FUNCTION_BLOCK FB_IndexedPatchPressMachine
VAR
    fbPatchFeedManager : FB_PatchFeedManager;
    bPatchDriveRunRequest : BOOL;
    bPatchSequenceAirRequest : BOOL;
    bPatchSequenceDownRequest : BOOL;
    bPatchHoldUpAllowed : BOOL;
    bPatchStartAllowed : BOOL;
    bPatchVerticalIndexReady : BOOL;
    bPatchVerticalUpCommandPrevious : BOOL;
    bPatchVerticalDownCommandPrevious : BOOL;
    fbIndex : FB_IndexTable4;
    fbMainDoorLock : FB_MainDoorLock;
    fbNestManager : FB_NestTableManager;
    fbOperatorStation : FB_OperatorStation;
    bOperatorLoadValid : BOOL;
    fbPatchDispense : FB_PatchDispenseStation;
    fbHeatStake : FB_HeatStakeStation;
    fbHeatStakeTemperature : FB_HeatStakeTemperatureControl;
    fbHeatStakePressureRegulator : FB_VeabPressureRegulator;
    fbVision : FB_VisionStation;
    fbVisionManualImages : FB_VisionManualImages;
    aVisionPbupReferenceKnown : ARRAY[1..4] OF BOOL;
    uiVisionPbupNest : UINT;
    uiVisionPbupEditNest : UINT;
    uiVisionImageOwnedNest : UINT;
    eVisionImageOwnedIndex : E_TablePosition;
    bVisionImagePermit : BOOL;
    bVisionImageJogBusy : BOOL;
    bVisionImageOwnedBeforeUpdate : BOOL;
    bVisionImageRecoveryRequired : BOOL;
    bManualImageTriggerCommand : BOOL;
    bManualCameraTransportReady : BOOL;
    bManualImageCameraFailed : BOOL;
    bVisionPbupFitted : BOOL;
    bVisionPbupKnown : BOOL;
    rtVisionPbupAutoBusy : R_TRIG;
    rtVisionPbupAutoDone : R_TRIG;
    tonVisionRotate0Confirm : TON;
    tonVisionRotate180Confirm : TON;
    tVisionRotaryConfirm : TIME := T#1S;
    bVisionRotate0Confirmed : BOOL;
    bVisionRotate180Confirmed : BOOL;
    bVisionRotate0CommandPrevious : BOOL;
    bVisionRotate180CommandPrevious : BOOL;
    bVisionTriggerAccepted : BOOL;
    bVisionRotatingCaptureAccepted : BOOL;
	fbVSCamera : FB_VSCamera;
    fbProcessCycle : FB_ProcessCycle;
    fbCommissioningGuard : FB_PatchPressCommissioningGuard;
    eMachineState : E_MachineState := E_MachineState.PowerUp;
    eInitialisingWaitReason : E_InitialisingWaitReason := E_InitialisingWaitReason.None;
    eStoppingWaitReason : E_StoppingWaitReason := E_StoppingWaitReason.None;
    stOutputsInternal : ST_MachineOutputs;
    stIndexStatus : ST_IndexStatus;
    stMainDoorStatus : ST_MainDoorLockStatus;
    stOperatorStatus : ST_OperatorStationStatus;
    stPatchDispenseStatus : ST_PatchStageStatus;
    stHeatStakeStatus : ST_PatchStageStatus;
    stHeatStakeTemperatureStatus : ST_HeatStakeTemperatureStatus;
    stHeatStakeProcessStatus : ST_HeatStakeProcessStatus;
    stVisionStatus : ST_PatchStageStatus;
    stOperatorNest : ST_Nest;
    stPatchDispenseNest : ST_Nest;
    stHeatStakeNest : ST_Nest;
    stHeatStakePresenceResult : ST_ProcessResult;
    stEmptyHeatStakePresenceResult : ST_ProcessResult;
    stVisionNest : ST_Nest;
	stPatchDispenseCycleResult : ST_ProcessResult;
    stHeatStakeCycleResult : ST_ProcessResult;

    bPatchDispenseRequired : BOOL;
    bHeatStakeRequired : BOOL;
    bVisionRequired : BOOL;
	
	bPatchHomeVerticalUpRequest : BOOL := FALSE;
	
	// Patch Dispensing Manual Mode
	bPatchManualEnableAllowed : BOOL;
	bPatchManualSupportAllowed : BOOL;
	bPatchManualVerticalAllowed : BOOL;
	bPatchManualAirAllowed : BOOL;

    // Snapshot taken before the station Update() calls.
    // Required to know which physical parts were actually being processed if
    // Safety is lost, because Update() immediately disables the station when
    // Safety_OK goes FALSE.
    bVisionProcessingBeforeUpdate 			: BOOL;

    // Machine-state transition tracking for one-shot product disposition.
    ePreviousMachineState 					: E_MachineState := E_MachineState.PowerUp;
    stProcessFaultResult 					: ST_ProcessResult;

    bAllRequiredStationsReady 				: BOOL;
    bAllRequiredStationsComplete 			: BOOL;
    bAnyStationInProcess 					: BOOL;
    bCycleResultsStored 					: BOOL;

    stPermissives 							: ST_MachinePermissives;
    tonInitialising 						: TON;
    tonStopping 							: TON;
	tonHeaterDwell 							: TON;

	
	
	bHeaterDwellTimeoutFault 				: BOOL := FALSE;
    bInitialisationTimeoutFault 			: BOOL;
    bStoppingTimeoutFault 					: BOOL;
    bAutoCycleAllowed 						: BOOL;
    sAutoCycleBlockReason 					: STRING(160);
    bIndexMoveAccepted 						: BOOL;
    bDoorLockOutput 						: BOOL;
	bMainDoorUnlockAcknowledged 			: BOOL := FALSE;
	bMainDoorHotLockRequired 				: BOOL := FALSE;
	
    rtManualIndexMove 						: R_TRIG;
	rtReprocessIndexAttempt 				: R_TRIG;
	rtMachineInitialising 					: R_TRIG;

    bProcessStartStations       			: BOOL;
    bProcessStopStations        			: BOOL;
    bProcessRequestIndex        			: BOOL;
    bProcessCycleActive         			: BOOL;
    bProcessCycleCompletePulse  			: BOOL;
    bProcessCycleFault          			: BOOL;
    bProcessCycleTimeoutFault   			: BOOL;
    bProcessStopPending         			: BOOL;
    bProcessAutomaticStopRequest 			: BOOL;
    bAutoCycleStopRequestLatched 			: BOOL;
    eProcessCycleState          			: E_CycleState;
    bDisabledNestIndexAttempt   			: BOOL;

    aNestSnapshot               			: ARRAY[1..4] OF ST_Nest;
    bDisabledNestPartPresent    			: BOOL;
    uiDisabledNestPartNestId    			: UINT;
    bDisabledNestPartPopupRequest 			: BOOL;
    uiDisabledNestPartPopupNestId 			: UINT;
    iNestCheck                  			: INT;

    // Reject chute full supervision / controlled stop.
    tonRejectChuteFull              : TON;
    tonRejectChutePopupReopen       : TON;
    rtRejectChuteAcknowledge        : R_TRIG;
    rtRejectChuteStopRequest        : R_TRIG;
    bRejectChuteFullLatched         : BOOL;
    bRejectChutePopupRequest        : BOOL;
    bRejectChuteStopRequestLatched  : BOOL;
    bRejectChutePopupReopenPending  : BOOL;
	bReprocessPopupAcknowledged 	: BOOL := FALSE;
	bReprocessAcknowledgePending 	: BOOL := FALSE;
	bHeaterDwellRequestLatched 		: BOOL := FALSE;

    // Manual controlled-stop tracking.
    bManualSupportTargetUpAtRejectStop : BOOL;
    bManualRejectStopReady             : BOOL;

    bStation1SupportExtendRequest  	: BOOL;
    bStation1SupportRetractRequest 	: BOOL;
    bStation2SupportExtendRequest  	: BOOL;
    bStation2SupportRetractRequest 	: BOOL;

    bHeatStakeHeadLockRequest 		: BOOL;
    bHeatStakeHeadUnlockRequest 	: BOOL;
    // Monostable valve output state; re-arm descent only after completed HOME.
    bHeatStakeHeadUpRecoveryLatched : BOOL := TRUE;
    bHeatStakeHeadDownHeld : BOOL := FALSE;
    bHeatStakeHeadDownRequest 		: BOOL;
    bHeatStakeHeadUpRequest 		: BOOL;
    rHeatStakePressureCommandBar 	: LREAL;
    iHeatStakePressureRaw 			: INT;
    rHeatStakePressureScaledBar 	: LREAL;
    bHeatStakeContactDwellActive 	: BOOL;
    usiHeatStakeSequenceStep 		: USINT;
	
	rtPatchSupportExtend 			: R_TRIG;
	rtPatchSupportRetract 			: R_TRIG;
	bPatchSupportExtendDesired 		: BOOL := FALSE;
	bPatchManualAllowed 			: BOOL;
	tpPatchAirBlow 					: TP;


    // Heat Stake Manual Mode
    rtHeatStakeManualStakePatch 	: R_TRIG;
    rtHeatStakeManualUnlock     	: R_TRIG;
    rtHeatStakeManualLock       	: R_TRIG;
    rtHeatStakeManualHeadDown   	: R_TRIG;
    rtHeatStakeManualHeadUp     	: R_TRIG;
    rtHeatStakeInitialising     	: R_TRIG;

    tonHeatStakeManualAction     	: TON;
    usiHeatStakeManualActionStep 	: USINT := 0;
    bHeatStakeManualHeadUnlocked 	: BOOL := FALSE;
    bHeatStakeManualStakeCycleActive : BOOL := FALSE;

    bHeatStakeStationHeadDownTimeoutFault 		: BOOL;
    bHeatStakeStationHeadUpTimeoutFault 		: BOOL;
    bHeatStakeStationHeadSensorConflictFault 	: BOOL;
    bHeatStakeManualHeadDownTimeoutFault 		: BOOL;
    bHeatStakeManualHeadUpTimeoutFault 			: BOOL;

    bHeatStakeManualEnableAllowed   : BOOL;
    bHeatStakeManualStakeAllowed    : BOOL;
    bHeatStakeManualUnlockAllowed   : BOOL;
    bHeatStakeManualLockAllowed     : BOOL;
    bHeatStakeManualHeadDownAllowed : BOOL;
    bHeatStakeManualHeadUpAllowed   : BOOL;
    bHeatStakeManualSupportAllowed  : BOOL;
    bHeatStakeManualActionBusy      : BOOL;
	
	// Vision Manual Mode

	tpVisionManualHorizontalBack  	: TP;
	tpVisionManualHorizontalFront 	: TP;
	


	
	rtVisionManualHorizontalBack  	: R_TRIG;
	rtVisionManualHorizontalFront 	: R_TRIG;
	rtVisionManualHome 				: R_TRIG;
	
	// Vision Manual - Vertical Intermediate


	
	bVisionManualVerticalUpActive 			: BOOL;

	bVisionManualVerticalFullDownActive     : BOOL;
	
	bVisionManualRotate0Active   			: BOOL;
	bVisionManualRotate180Active 			: BOOL;

    // Manual Heat Stake tooling-position tracking uses physical sensors.
    bHeatStakeManualHomePosition     		: BOOL;
    bHeatStakeManualOutOfHome        		: BOOL;

    bVisionHorizontalBackRequest  : BOOL;
    bVisionHorizontalFrontRequest : BOOL;
    bVisionVerticalUpRequest      : BOOL;
    bVisionVerticalDownRequest    : BOOL;

    bVisionGripCloseRequest       : BOOL;
    bVisionGripOpenRequest        : BOOL;
    bVisionRotate0Request         : BOOL;
    bVisionRotate180Request       : BOOL;
	
	//CAMERA
	bVisionTriggerRequest			: BOOL;
	bVisionChangeProgramRequest		: BOOL;
	bVisionGetResultsRequest		: BOOL;
	bVisionGetResultsReadyRequest	: BOOL;
	bVisionResetResultsRequest		: BOOL;
	bVisionAcknowledgeResultsRquest	: BOOL;
	nVisionProgramNumber			: UDINT;
	bVisionGetCurrentProgram		: UDINT;
	
	nVisionResults					: ST_VisionResults;
    rtVisionCameraResultsReset : R_TRIG;
	
		
		// Vision Manual Mode
	bVisionManualEnableAllowed          : BOOL;
    bVisionCameraStartBlocked : BOOL; // Live camera error/recovery latch; blocks new starts.
	
	bVisionHorizontalBackAllowed        : BOOL;
	bVisionHorizontalFrontAllowed       : BOOL;
	
	bVisionVerticalUpAllowed            : BOOL;

	bVisionVerticalFullDownAllowed      : BOOL;
	
	bVisionGripOpenAllowed              : BOOL;
	bVisionGripCloseAllowed             : BOOL;
	
	bVisionRotate0Allowed               : BOOL;
	bVisionRotate180Allowed             : BOOL;
	
	bVisionManualRunSequenceAllowed 	: BOOL;
	bVisionManualSequenceActive 		: BOOL;
	bVisionManualHomeAllowed 			: BOOL;
	bVisionManualHomeActive  			: BOOL;

// Already existed:
// bVisionSupportAllowed : BOOL;
    // Fault reset is latched because PRG_Events executes after PRG_Main.
    // The event manager may clear its fault latch on the same Reset scan,
    // therefore the machine must remember the request until the following scan.
    bFaultResetRequested 				: BOOL;
    bAirAndDoorEnable 					: BOOL;
    // Air can only be latched ON by System Initialising.
    // Once ON, it may remain ON through Stopping/Stopped while the main door
    // stays closed. Opening the door, or entering Fault, clears this latch.
    bAirSupplyLatched 					: BOOL;
    // PLC-originated machine faults pulse the TwinSAFE Run/Stop request low.
    // RunRequest is otherwise TRUE so TwinSAFE can execute and return Safety_OK.
    bSafetyDropRequest 					: BOOL;
    tpSafetyRunDrop 					: TP;
    tonLedBlink 						: TON;
    rtLedBlink 							: R_TRIG;
	
	tonHMIAliveOn  						: TON;
	tonHMIAliveOff 						: TON;
	bOutHMI        						: BOOL := TRUE;
	
	
	
    bLedBlinkState : BOOL;
	
	btest								: ARRAY [1..10] OF BOOL;
	ntest								: UDINT;
	
	sHeaterMinimum 						: STRING(32);
	sHeaterCurrent 						: STRING(32);
	
	// =====================================================
	// PATCH DISPENSING - MANUAL VERTICAL
	// =====================================================
    bPatchManualVerticalUpHeld : BOOL := TRUE; // Retain the selected UP direction while manual control is permitted.
    bPatchManualVerticalDownHeld : BOOL; // Retain the selected DOWN direction while manual control is permitted.
	
	bPatchVerticalUpAllowed   : BOOL;
	bPatchVerticalDownAllowed : BOOL;
	
	tonPatchHomeUpOutputVerify : TON;
	bPatchHomeUpOutputVerified : BOOL := FALSE;
	
    // Per-product volatile confidence/location; existing retained fitted array stays compatible.
    aVisionProductLocation : ARRAY[1..4] OF USINT; // 0 unknown, 1 nest, 2 legacy nest alias, 3 held; PBUP state is separate.
    aVisionPbupSource : ARRAY[1..4] OF USINT;
    aVisionLoadEmptySeen : ARRAY[1..4] OF BOOL;
    aVisionLoadCandidate : ARRAY[1..4] OF BOOL;
    uiVisionLoadObservedNest : UINT;
    tonVisionLoadEmpty : TON;
    tonVisionLoadPair : TON;
    bManualIndexAttempt : BOOL;
    bManualIndexStartAllowed : BOOL;
    bManualIndexWarningActive : BOOL;
    bManualIndexBlockVision : BOOL;
    bManualIndexBlockHeat : BOOL;
    bManualIndexBlockPatch : BOOL;
    bManualIndexBlockOther : BOOL;
    bManualCameraDrainResult : BOOL;
    bManualCameraDiscardedResult : BOOL;
    stManualCameraDiscardedResults : ST_VisionResults;
    bManualCameraRecoveryAllowed : BOOL;
    bManualCameraRecoveryActive : BOOL;
    bManualCameraRecoveryFailed : BOOL;
    bManualCameraCaptureAfterRecovery : BOOL;
    bManualCameraClearError0 : BOOL;
    bManualCameraClearError1 : BOOL;
    usiManualCameraRecoveryStep : USINT;
    udiManualCameraRecoveryImage : UDINT;
    udiManualCameraRecoveryError0 : UDINT;
    udiManualCameraRecoveryError1 : UDINT;
    tonManualCameraRecovery : TON;
    sManualCameraRecoveryMessage : STRING(160);
    bManualCameraResetOnly : BOOL;
    bManualCameraRecoveredPulse : BOOL;
END_VAR
VAR
    bManualCameraAllowed : BOOL;
    bManualCameraOwner : BOOL;
    bManualCameraReset : BOOL;
    bManualCameraConsume : BOOL;
    usiManualCameraStep : USINT;
    udiManualCameraProgram : UDINT;
    udiManualCameraSelection : UDINT;
    stManualCameraResults : ST_VisionResults;
    tonManualCamera : TON;
END_VAR

METHOD PUBLIC Cyclic
VAR_INPUT
    stInputs : ST_MachineInputs;
    stCommand : ST_MachineCommand;
    stConfig : ST_MachineConfig;
    stHeatStakeTemperatureSettings : ST_HeatStakeTemperatureSettings;
    stHeatStakeProcessSettings : ST_HeatStakeProcessSettings;
    bPatchDispenseCommissioned : BOOL;
    bHeatStakeCommissioned : BOOL;
    bVisionCommissioned : BOOL;
    bCoreCommissioningMode : BOOL;
    bLogoutHMI : BOOL;
	
	
	
	
END_VAR
VAR_OUTPUT
    stOutputs : ST_MachineOutputs;
    stStatus : ST_MachineStatus;
END_VAR
tVisionRotaryConfirm := UDINT_TO_TIME(GVL_Persistent.stVisionProcessSettings.udiRotaryConfirmMs);
ResetCyclicOutputs();

// Shared endpoint interpretation for automatic, HOME, Manual and HMI.
tonVisionRotate0Confirm(IN := bVisionCommissioned AND stInputs.stSafety.bSafetyOk
    AND GVL_Safety.bAirSupplySafe AND NOT stCommand.bReset
    AND stInputs.bRotaryGripperPick0 AND NOT stInputs.bRotaryGripperPlace180
    AND NOT bVisionRotate180CommandPrevious
    AND (bVisionRotate0CommandPrevious OR bVisionRotate0Confirmed), PT := tVisionRotaryConfirm);
tonVisionRotate180Confirm(IN := bVisionCommissioned AND stInputs.stSafety.bSafetyOk
    AND GVL_Safety.bAirSupplySafe AND NOT stCommand.bReset
    AND stInputs.bRotaryGripperPlace180 AND NOT stInputs.bRotaryGripperPick0
    AND NOT bVisionRotate0CommandPrevious, PT := tVisionRotaryConfirm);
bVisionRotate0Confirmed := tonVisionRotate0Confirm.Q;
bVisionRotate180Confirmed := tonVisionRotate180Confirm.Q;


// Air-memory rule:
// - only Initialising may set bAirSupplyLatched TRUE;
// - an open main door always clears it immediately;
// - therefore air can never remain ON with the door open;
// - closing the door again does NOT restore air unless a new Initialising
//   sequence is entered.
IF NOT stInputs.bMainDoorClosed THEN
    bAirSupplyLatched := FALSE;
END_IF


	
	// =====================================================
	// HEATER DWELL TIMEOUT SUPERVISION
	// =====================================================
	// Timer runs only while the machine is in Dwell.
	// Leaving Dwell automatically resets the timer.
	
	tonHeaterDwell(
		IN := (eMachineState = E_MachineState.Dwell),
		PT := stConfig.tHeaterDwellTimeout
	);
	
	// Latch the timeout fault until machine Reset.
	IF tonHeaterDwell.Q THEN
		bHeaterDwellTimeoutFault := TRUE;
	END_IF
	
	// Clear the latched Heater Dwell timeout fault
	// when the operator requests Reset from Fault.
	
	IF stCommand.bReset
		AND (eMachineState = E_MachineState.Fault)
	THEN
		bHeaterDwellTimeoutFault := FALSE;
	END_IF

// One-scan internal request. A PLC machine fault sets this TRUE below;
// TP converts it into a deterministic TwinSAFE Run/Stop drop pulse.
bSafetyDropRequest := FALSE;

// =========================================================
// REJECT CHUTE FULL SUPERVISION
// =========================================================
// The reject chute sensor can pulse briefly during a normal reject.
// Only a continuous TRUE for 2 seconds means CHUTE FULL.
tonRejectChuteFull(
    IN := stInputs.bRejectChutePartPresent,
    PT := T#2S
);

rtRejectChuteAcknowledge(
    CLK := stCommand.bAcknowledgeRejectChuteFull
);

// First confirmed full condition:
// - latch operator intervention;
// - request popup;
// - latch a controlled Stop Request.
IF tonRejectChuteFull.Q
    AND NOT bRejectChuteFullLatched
THEN
    bRejectChuteFullLatched := TRUE;
    bRejectChutePopupRequest := TRUE;
    bRejectChuteStopRequestLatched := TRUE;
END_IF

// Acknowledge is only valid for clearing the interlock when the physical
// sensor is already FALSE.
IF rtRejectChuteAcknowledge.Q
    AND bRejectChuteFullLatched
THEN
    IF NOT stInputs.bRejectChutePartPresent THEN
        bRejectChuteFullLatched := FALSE;
        bRejectChutePopupRequest := FALSE;
        bRejectChutePopupReopenPending := FALSE;
    ELSE
        // Operator acknowledged while still full: close briefly, then reopen.
        bRejectChutePopupRequest := FALSE;
        bRejectChutePopupReopenPending := TRUE;
    END_IF
END_IF

tonRejectChutePopupReopen(
    IN := bRejectChutePopupReopenPending,
    PT := T#500MS
);

IF tonRejectChutePopupReopen.Q THEN
    bRejectChutePopupReopenPending := FALSE;
    IF bRejectChuteFullLatched THEN
        bRejectChutePopupRequest := TRUE;
    END_IF
END_IF

// Capture Manual support target at the instant the controlled stop is first
// requested. If it is already travelling, allow that existing stroke to finish.
rtRejectChuteStopRequest(
    CLK := bRejectChuteStopRequestLatched
);

IF rtRejectChuteStopRequest.Q
    AND (eMachineState = E_MachineState.Manual)
THEN
    bManualSupportTargetUpAtRejectStop :=
        stCommand.bHeatStakeManualSupportUp;
END_IF


// 500 ms operator indication blink, matching the validated Silicone core.
tonLedBlink(IN := NOT tonLedBlink.Q, PT := T#500MS);
rtLedBlink(CLK := tonLedBlink.Q);
IF rtLedBlink.Q THEN
    bLedBlinkState := NOT bLedBlinkState;
END_IF

// Heat Stake temperature preheat/control.
fbHeatStakeTemperature.Cyclic(
    bEnable :=
        (eMachineState = E_MachineState.ReadyToStart)
		OR (eMachineState = E_MachineState.Dwell)
        OR (eMachineState = E_MachineState.AutoCycle)
        OR (
            (eMachineState = E_MachineState.Manual)
            AND (
                stCommand.bHeatStakeManualEnable
                OR bHeatStakeManualStakeCycleActive
            )
        ),
    bAutoCycleActive := (eMachineState = E_MachineState.AutoCycle),
    bSafetyOk := stInputs.stSafety.bSafetyOk,
    diTc1Raw := stInputs.diHeatStakeTc1Raw,
    diTc2Raw := stInputs.diHeatStakeTc2Raw,
    diTc3Raw := stInputs.diHeatStakeTc3Raw,
    stSettings := stHeatStakeTemperatureSettings,
    uiPwm1Raw => stOutputsInternal.uiHeatStakePwm1Raw,
    uiPwm2Raw => stOutputsInternal.uiHeatStakePwm2Raw,
    stStatus => stHeatStakeTemperatureStatus
);


	// =====================================================
	// HEATER LOW TEMPERATURE - DWELL REQUEST
	// =====================================================
	// Latch the request when temperature drops during AutoCycle.
	// The current station processes must finish before entering Dwell.
	
	IF (eMachineState = E_MachineState.AutoCycle)
		AND NOT stHeatStakeTemperatureStatus.bIndexTemperatureReady
		AND NOT stHeatStakeTemperatureStatus.bFault
	THEN
		bHeaterDwellRequestLatched := TRUE;
	END_IF
	
	// =====================================================
	// HEATER DWELL - REQUEST RESET
	// =====================================================
	// Preserve the request while AutoCycle is completing
	// the current production cycle.
	//
	// Clear it if the machine leaves the automatic
	// production sequence through Stop or Fault.
	
	IF (eMachineState = E_MachineState.Stopping)
		OR (eMachineState = E_MachineState.Stopped)
		OR (eMachineState = E_MachineState.Fault)
	THEN
		bHeaterDwellRequestLatched := FALSE;
	END_IF

//Camera
//---------------------------------------------------------------------------------------------------
fbVSCamera(
    stCameraIO := GVL_EtherCAT.stVSKeyenceCamera,
    udiError0Code := GVL_EtherCAT.udiVisionError0Code,
    udiError1Code := GVL_EtherCAT.udiVisionError1Code,
    bResetRequest := stCommand.bReset
);
bVisionGetCurrentProgram := fbVSCamera.GetCurrentProgram();

// Sample the physical edge even when disabled/blocked. Never create an edge on Enable.
rtManualIndexMove(CLK := stInputs.bTwoHandsSafe);
bManualIndexAttempt := rtManualIndexMove.Q AND (eMachineState = E_MachineState.Manual)
    AND stCommand.bIndexerManualEnable AND NOT bRejectChuteStopRequestLatched;

// Manual camera commands are consumed once; camera output ownership remains here.
GVL_HMI.bCameraConnected := (GVL_EtherCAT.wVisionPnState = 0)
    AND (GVL_EtherCAT.wVisionPnDiag = 2)
    AND GVL_EtherCAT.stTerm22_EL6633.stTerminalInfo.bTerminalOperational;
bManualCameraAllowed := (eMachineState = E_MachineState.Manual)
    AND stCommand.bVisionManualEnable AND stInputs.stSafety.bSafetyOk
    AND (GVL_EtherCAT.stVSKeyenceCamera.bRunStatus OR fbVSCamera.IsFaulted()
        OR bManualCameraRecoveryActive OR bVisionCameraStartBlocked
        OR fbVisionManualImages.bPrepared OR (fbVisionManualImages.usiStep = 210)
        OR fbVisionManualImages.bCameraWarning)
    AND NOT stCommand.bStop AND NOT stCommand.bReset
    AND (fbVisionManualImages.bActive
        OR (NOT stCommand.bVisionManualRunSequence AND NOT stCommand.bVisionManualHomeRequest))
    AND stInputs.bMainDoorClosed AND GVL_Safety.bAirSupplySafe
    AND bVisionCommissioned AND NOT stInputs.bEventFault
    AND NOT stInputs.bEventCycleStopRequest AND NOT bRejectChuteStopRequestLatched
    AND stInputs.bIndexReady AND stInputs.bIndexLocked AND NOT stIndexStatus.bBusy
    AND (stInputs.eIndexPosition <> E_TablePosition.Unknown)
    AND (NOT fbVision.IsBusy() OR fbVisionManualImages.bActive)
    AND NOT fbVisionManualImages.bFault
    AND NOT bVisionManualSequenceActive AND NOT bVisionManualHomeActive;
GVL_HMI.bCameraResetAllowed := (eMachineState = E_MachineState.Manual)
    AND stCommand.bVisionManualEnable AND stInputs.stSafety.bSafetyOk
    AND stInputs.bMainDoorClosed AND GVL_Safety.bAirSupplySafe AND GVL_HMI.bCameraConnected
    AND NOT stCommand.bStop AND NOT stCommand.bReset AND NOT stInputs.bEventFault
    AND NOT stInputs.bEventCycleStopRequest AND NOT bRejectChuteStopRequestLatched
    AND stInputs.bIndexReady AND stInputs.bIndexLocked AND NOT stIndexStatus.bBusy
    AND (stInputs.eIndexPosition <> E_TablePosition.Unknown)
    AND NOT bVisionManualSequenceActive AND NOT bVisionManualHomeActive
    AND (usiManualCameraStep = 0) AND NOT bManualCameraRecoveryActive
    AND NOT fbVisionManualImages.bBusy AND NOT bVisionImageJogBusy
    AND NOT stInputs.bTwoHandsSafe AND NOT stIndexStatus.bTwoHandRequired;
bManualCameraOwner := (bManualCameraAllowed
    AND (GVL_HMI.udiCameraManualImageSelection >= 1) AND (GVL_HMI.udiCameraManualImageSelection <= 4))
    OR (GVL_HMI.bCameraReset AND GVL_HMI.bCameraResetAllowed)
    OR (bManualCameraRecoveryActive AND (eMachineState = E_MachineState.Manual)
        AND stInputs.stSafety.bSafetyOk AND stInputs.bMainDoorClosed AND GVL_Safety.bAirSupplySafe
        AND GVL_HMI.bCameraConnected AND NOT stCommand.bStop AND NOT stCommand.bReset
        AND NOT stInputs.bEventFault AND NOT stInputs.bEventCycleStopRequest
        AND NOT bRejectChuteStopRequestLatched);
bManualImageTriggerCommand := GVL_HMI.bCameraManualTrigger;
bManualImageCameraFailed := FALSE;
bManualCameraRecoveredPulse := FALSE;
bManualCameraReset := FALSE;
bManualCameraConsume := FALSE;
tonManualCamera(IN := (usiManualCameraStep <> 0), PT := T#10S);
// An explicit operator click may recover camera errors. No reset/GoToRun/motion.
// A click at an already prepared position requests ONE capture after recovery.
// At HOME without a prepared image it recovers only; Prepare is still required.
bManualCameraRecoveryAllowed := bManualCameraOwner
    AND (bVisionCameraStartBlocked OR fbVisionManualImages.bCameraWarning)
    AND GVL_HMI.bCameraConnected AND (usiManualCameraStep = 0)
    AND NOT bManualCameraRecoveryActive AND NOT fbVisionManualImages.bFault
    AND NOT fbVisionManualImages.bBusy AND NOT bVisionImageJogBusy
    AND (fbVisionManualImages.bPrepared OR stVisionStatus.bHome)
    AND NOT stInputs.bTwoHandsSafe AND NOT stIndexStatus.bTwoHandRequired;
IF (bManualImageTriggerCommand AND bManualCameraRecoveryAllowed)
    OR (GVL_HMI.bCameraReset AND GVL_HMI.bCameraResetAllowed) THEN
    bManualCameraResetOnly := GVL_HMI.bCameraReset;
    bManualCameraRecoveryActive := TRUE;
    bManualCameraRecoveryFailed := FALSE;
    usiManualCameraRecoveryStep := 1;
    udiManualCameraRecoveryImage := GVL_HMI.udiCameraManualImageSelection;
    IF bManualCameraResetOnly THEN
        udiManualCameraRecoveryImage := GVL_EtherCAT.stVSKeyenceCamera.bCurrentProgramNumber + 1;
    END_IF
    bManualCameraCaptureAfterRecovery := NOT bManualCameraResetOnly AND fbVisionManualImages.bPrepared
        AND (fbVisionManualImages.udiPreparedImage = udiManualCameraRecoveryImage)
        AND bVisionPbupKnown;
    bManualCameraClearError0 := GVL_EtherCAT.stVSKeyenceCamera.abError[1];
    bManualCameraClearError1 := GVL_EtherCAT.stVSKeyenceCamera.abError[2];
    udiManualCameraRecoveryError0 := GVL_EtherCAT.udiVisionError0Code;
    udiManualCameraRecoveryError1 := GVL_EtherCAT.udiVisionError1Code;
    // Discard only the old software camera transaction. Live error feedback stays visible.
    bManualCameraReset := TRUE;
END_IF
tonManualCameraRecovery(IN := bManualCameraRecoveryActive, PT := T#3S);
IF bManualCameraRecoveryActive THEN
    bManualImageTriggerCommand := FALSE;
    IF NOT bManualCameraOwner OR NOT GVL_HMI.bCameraConnected
        OR (NOT bManualCameraResetOnly AND (GVL_HMI.udiCameraManualImageSelection <> udiManualCameraRecoveryImage))
        OR bVisionImageJogBusy OR stCommand.bStop OR stCommand.bReset
        OR (bManualCameraCaptureAfterRecovery AND NOT fbVisionManualImages.bPrepared) THEN
        bManualCameraRecoveryActive := FALSE;
        bManualCameraCaptureAfterRecovery := FALSE;
        bManualCameraRecoveryFailed := TRUE;
        sManualCameraRecoveryMessage := 'Camera recovery cancelled; no capture sent';
    ELSIF tonManualCameraRecovery.Q THEN
        bManualCameraRecoveryActive := FALSE;
        bManualCameraCaptureAfterRecovery := FALSE;
        bManualCameraRecoveryFailed := TRUE;
        sManualCameraRecoveryMessage := 'Camera recovery timeout; check camera, then retry';
    ELSIF (GVL_EtherCAT.stVSKeyenceCamera.abError[1]
            AND (NOT bManualCameraClearError0 OR (GVL_EtherCAT.udiVisionError0Code <> udiManualCameraRecoveryError0)))
        OR (GVL_EtherCAT.stVSKeyenceCamera.abError[2]
            AND (NOT bManualCameraClearError1 OR (GVL_EtherCAT.udiVisionError1Code <> udiManualCameraRecoveryError1))) THEN
        bManualCameraRecoveryActive := FALSE;
        bManualCameraCaptureAfterRecovery := FALSE;
        bManualCameraRecoveryFailed := TRUE;
        sManualCameraRecoveryMessage := 'Camera error changed; inspect camera before retry';
    ELSIF usiManualCameraRecoveryStep = 1 THEN
        sManualCameraRecoveryMessage := 'Camera: requesting error clear';
        IF NOT GVL_EtherCAT.stVSKeyenceCamera.abError[1]
            AND NOT GVL_EtherCAT.stVSKeyenceCamera.abError[2] THEN
            usiManualCameraRecoveryStep := 2;
        END_IF
    ELSE
        sManualCameraRecoveryMessage := 'Camera: waiting for RUN / clean handshake';
        IF GVL_EtherCAT.stVSKeyenceCamera.bRunStatus
            AND GVL_EtherCAT.stVSKeyenceCamera.bTriggerReady
            AND NOT GVL_EtherCAT.stVSKeyenceCamera.bTriggerAcknowledge
            AND NOT GVL_EtherCAT.stVSKeyenceCamera.bResultsReady
            AND NOT GVL_EtherCAT.stVSKeyenceCamera.bResultAck
            AND NOT GVL_EtherCAT.stVSKeyenceCamera.bProgramLoadExecute
            AND (GVL_EtherCAT.stVSKeyenceCamera.bCurrentProgramNumber = udiManualCameraRecoveryImage - 1) THEN
            bManualCameraRecoveryActive := FALSE;
            bManualCameraRecoveryFailed := FALSE;
            bManualCameraRecoveredPulse := TRUE;
            bManualImageTriggerCommand := bManualCameraCaptureAfterRecovery;
            bManualCameraCaptureAfterRecovery := FALSE;
            sManualCameraRecoveryMessage := 'Camera recovered; prepare if no position is reserved';
        END_IF
    END_IF
END_IF

GVL_HMI.bCameraReset := FALSE; // Accepted or rejected once, never queued.
IF NOT bManualCameraRecoveryActive THEN bManualCameraResetOnly := FALSE; END_IF
IF NOT bManualCameraOwner THEN
    IF usiManualCameraStep <> 0 THEN bManualCameraReset := TRUE; END_IF
    usiManualCameraStep := 0;
    GVL_HMI.bCameraManualPass := FALSE;
    GVL_HMI.bCameraManualFail := FALSE;
    GVL_HMI.sCameraManualMessage := 'Select an image in enabled Vision Manual mode';
ELSE
    IF (udiManualCameraSelection <> GVL_HMI.udiCameraManualImageSelection) AND (usiManualCameraStep = 0) THEN
        udiManualCameraSelection := GVL_HMI.udiCameraManualImageSelection;
        GVL_HMI.bCameraManualPass := FALSE;
        GVL_HMI.bCameraManualFail := FALSE;
    END_IF
    IF fbVisionManualImages.bActive AND fbVisionManualImages.bCaptureRequest
        AND (usiManualCameraStep = 0)
        AND GVL_HMI.bCameraConnected AND GVL_EtherCAT.stVSKeyenceCamera.bRunStatus
        AND NOT fbVSCamera.IsFaulted() THEN
        udiManualCameraProgram := fbVisionManualImages.udiPreparedImage - 1;
        usiManualCameraStep := 10;
        bManualCameraReset := TRUE;
        GVL_HMI.bCameraManualPass := FALSE;
        GVL_HMI.bCameraManualFail := FALSE;
        GVL_HMI.sCameraManualMessage := 'Loading selected program';
    END_IF
    IF usiManualCameraStep <> 0 THEN
        IF fbVisionManualImages.bCameraWarning
            OR NOT GVL_HMI.bCameraConnected OR NOT GVL_EtherCAT.stVSKeyenceCamera.bRunStatus
            OR fbVSCamera.IsFaulted() OR fbVSCamera.bRecoveryFailed OR tonManualCamera.Q THEN
            usiManualCameraStep := 0;
            bManualCameraReset := TRUE;
            bManualImageCameraFailed := TRUE;
            GVL_HMI.sCameraManualMessage := 'Capture aborted: connection, Run, camera error or timeout';
        ELSIF (usiManualCameraStep = 10)
            AND (GVL_EtherCAT.stVSKeyenceCamera.bCurrentProgramNumber = udiManualCameraProgram)
            AND NOT GVL_EtherCAT.stVSKeyenceCamera.bProgramLoadExecute THEN
            usiManualCameraStep := 20;
            GVL_HMI.sCameraManualMessage := 'Waiting for capture';
        ELSIF (usiManualCameraStep = 30)
            AND NOT GVL_EtherCAT.stVSKeyenceCamera.bResultsReady
            AND NOT GVL_EtherCAT.stVSKeyenceCamera.bTriggerAcknowledge THEN
            usiManualCameraStep := 0;
        END_IF
    END_IF
END_IF
GVL_HMI.bCameraManualTrigger := FALSE;
IF bManualCameraOwner THEN
    IF (usiManualCameraStep = 0) AND bManualCameraResetOnly THEN
        udiManualCameraProgram := udiManualCameraRecoveryImage - 1;
    ELSIF (usiManualCameraStep = 0) AND (GVL_HMI.udiCameraManualImageSelection >= 1)
        AND (GVL_HMI.udiCameraManualImageSelection <= 4) THEN
        udiManualCameraProgram := GVL_HMI.udiCameraManualImageSelection - 1;
    END_IF
END_IF

// Reset the accumulated payload before sampling any result in the new cycle.
rtVisionCameraResultsReset(CLK := (stVisionStatus.eState = E_PatchStationState.Processing));
IF bManualCameraReset OR bVisionResetResultsRequest OR rtVisionCameraResultsReset.Q THEN
    fbVSCamera.GetResults(stVisionResults => nVisionResults, bResetResults := TRUE);
END_IF

// Apply previous-scan station commands, then sample ACK/result in this scan.
// Close an unacknowledged moving-picture request at the physical 180 end sensor.
IF (bManualCameraOwner AND (usiManualCameraStep = 0))
    OR (NOT bManualCameraOwner AND NOT bVisionTriggerRequest) THEN
    bVisionRotatingCaptureAccepted := FALSE;
END_IF
bVisionTriggerAccepted := fbVSCamera.RequestTrigger(
    bEnable := (bManualCameraOwner AND (usiManualCameraStep = 20)
        AND ((udiManualCameraProgram <> 1) OR NOT fbVisionManualImages.bMovingCapture
            OR NOT stInputs.bRotaryGripperPlace180 OR bVisionRotatingCaptureAccepted
            OR GVL_EtherCAT.stVSKeyenceCamera.bTriggerAcknowledge))
        OR (NOT bManualCameraOwner AND bVisionTriggerRequest
        AND ((GVL_EtherCAT.stVSKeyenceCamera.bCurrentProgramNumber <> 1)
            OR NOT stInputs.bRotaryGripperPlace180
            OR bVisionRotatingCaptureAccepted
            OR GVL_EtherCAT.stVSKeyenceCamera.bTriggerAcknowledge)));
IF bVisionTriggerAccepted AND (GVL_EtherCAT.stVSKeyenceCamera.bCurrentProgramNumber = 1) THEN
    bVisionRotatingCaptureAccepted := TRUE;
END_IF
IF bManualCameraOwner THEN
    fbVSCamera.RequestChangeProgram(bEnable := NOT bManualCameraResetOnly, nProgramNumber := udiManualCameraProgram);
ELSE
    fbVSCamera.RequestChangeProgram(bEnable := bVisionChangeProgramRequest, nProgramNumber := nVisionProgramNumber);
END_IF
fbVSCamera.Cyclic();
// A pre-existing camera error must be visible before a new station attempt.
bVisionCameraStartBlocked := fbVSCamera.IsFaulted() OR fbVSCamera.bRecoveryFailed;
bVisionGetResultsReadyRequest := fbVSCamera.GetResultsReady();
IF bManualCameraOwner AND (usiManualCameraStep = 20) AND bVisionGetResultsReadyRequest THEN
    bManualCameraConsume := fbVSCamera.GetResults(stVisionResults => stManualCameraResults, bResetResults := FALSE);
    IF bManualCameraConsume THEN
        GVL_HMI.bCameraManualPass := stManualCameraResults.aInspectionCompleted[udiManualCameraProgram + 1]
            AND stManualCameraResults.aInspectionPassed[udiManualCameraProgram + 1];
        GVL_HMI.bCameraManualFail := stManualCameraResults.aInspectionCompleted[udiManualCameraProgram + 1]
            AND NOT stManualCameraResults.aInspectionPassed[udiManualCameraProgram + 1];
        GVL_HMI.udiCameraManualCaptureCount := GVL_HMI.udiCameraManualCaptureCount + 1;
        GVL_HMI.sCameraManualMessage := 'Capture complete';
        usiManualCameraStep := 30;
    END_IF
END_IF
GVL_HMI.bCameraManualAllowed := bManualCameraAllowed;
GVL_HMI.bCameraManualBusy := bManualCameraRecoveryActive OR (usiManualCameraStep <> 0)
    OR (bManualCameraOwner AND GVL_HMI.bCameraConnected AND GVL_EtherCAT.stVSKeyenceCamera.bRunStatus
        AND (GVL_EtherCAT.stVSKeyenceCamera.bCurrentProgramNumber <> udiManualCameraProgram));
bManualCameraTransportReady := bManualCameraOwner AND GVL_HMI.bCameraConnected
    AND GVL_EtherCAT.stVSKeyenceCamera.bRunStatus AND NOT fbVSCamera.IsFaulted()
    AND NOT fbVSCamera.bRecoveryFailed AND NOT GVL_HMI.bCameraManualBusy
    AND (GVL_EtherCAT.stVSKeyenceCamera.bCurrentProgramNumber = udiManualCameraProgram)
    AND GVL_EtherCAT.stVSKeyenceCamera.bTriggerReady
    AND NOT GVL_EtherCAT.stVSKeyenceCamera.bTriggerAcknowledge
    AND NOT GVL_EtherCAT.stVSKeyenceCamera.bResultsReady
    AND NOT GVL_EtherCAT.stVSKeyenceCamera.bResultAck
    AND NOT bManualCameraRecoveryActive;


IF NOT bManualCameraOwner AND bVisionGetResultsRequest
    AND NOT bVisionResetResultsRequest
    AND NOT rtVisionCameraResultsReset.Q THEN
    fbVSCamera.GetResults(stVisionResults => nVisionResults, bResetResults := FALSE);
END_IF

bManualCameraDrainResult := FALSE;
IF bManualCameraOwner AND (usiManualCameraStep = 0)
    AND NOT fbVisionManualImages.bBusy AND NOT fbVisionManualImages.bCaptureRequest
    AND NOT fbVSCamera.IsFaulted() AND NOT fbVSCamera.bRecoveryFailed THEN
    bManualCameraDiscardedResult := fbVSCamera.GetResults(
        stVisionResults => stManualCameraDiscardedResults, bResetResults := FALSE);
    bManualCameraDrainResult := GVL_EtherCAT.stVSKeyenceCamera.bResultsReady
        OR bManualCameraDiscardedResult;
END_IF

// Copy the latched payload before acknowledging/releasing it.
IF bManualCameraDrainResult OR (bManualCameraOwner AND (usiManualCameraStep = 30))
    OR (NOT bManualCameraOwner AND bVisionAcknowledgeResultsRquest
        AND bVisionGetResultsRequest
        AND NOT bVisionResetResultsRequest
        AND NOT rtVisionCameraResultsReset.Q) THEN
    fbVSCamera.RequestResultsAck(bEnable := TRUE);
ELSE
    fbVSCamera.RequestResultsAck(bEnable := FALSE);
END_IF
// Explicit operator recovery is the only manual owner of these clear outputs.
// FB_VSCamera.Cyclic defaults them FALSE each scan; never clear a new/different error.
IF bManualCameraRecoveryActive AND (usiManualCameraRecoveryStep = 1) THEN
    GVL_EtherCAT.stVSKeyenceCamera.abErrorClear[1] := bManualCameraClearError0
        AND GVL_EtherCAT.stVSKeyenceCamera.abError[1];
    GVL_EtherCAT.stVSKeyenceCamera.abErrorClear[2] := bManualCameraClearError1
        AND GVL_EtherCAT.stVSKeyenceCamera.abError[2];
END_IF
IF bManualCameraTransportReady THEN bManualCameraRecoveryFailed := FALSE; END_IF
GVL_MASTER.bManualCameraRecoveryFailed := bManualCameraRecoveryFailed;
//---------------------------------------------------------------------------------------------------

// Patch feeding owns its axis commands; it does not own physical safety outputs.
// Stopping withdraws M1 control. FB_PatchFeedAxis retains power for its own
// controlled halt; do not start a previously idle M1 simply by entering Stopping.
fbPatchFeedManager.Cyclic(
    bDrivePermit := bPatchDispenseCommissioned AND stInputs.bMainDoorClosed
        AND GVL_Safety.bAirSupplySafe AND NOT stInputs.bEventFault
        AND ((eMachineState = E_MachineState.AutoCycle)
            OR ((eMachineState = E_MachineState.Manual)
                AND (stCommand.bPatchManualEnable OR fbPatchDispense.IsBusy()))),
    bDriveRunRequest := bPatchDriveRunRequest,
    bPermit := bPatchDispenseCommissioned
        AND ((eMachineState = E_MachineState.AutoCycle)
            OR ((eMachineState = E_MachineState.Manual) AND stCommand.bPatchManualEnable))
        AND stInputs.bMainDoorClosed AND GVL_Safety.bAirSupplySafe
        AND NOT stCommand.bStop AND NOT stInputs.bEventFault
        AND NOT stInputs.bEventCycleStopRequest
        AND NOT bRejectChuteStopRequestLatched AND NOT bAutoCycleStopRequestLatched,
    bSafetyOk := stInputs.stSafety.bMotionSafetyPermitted,
    bReset := stCommand.bReset,
    bMiddleDown := stInputs.bMiddleRockerDown,
    bMiddleUp := stInputs.bMiddleRockerUp,
    bTopDown := stInputs.bTopRockerDown,
    bTopUp := stInputs.bTopRockerUp,
    bPatchFeedStart := stInputs.bBottomRockerUp, // Term19 Input14
    bPatchFeedStop := stInputs.bBottomRockerDown, // Term19 Input13
    stSettings := GVL_Motion.stPatchFeedSettings,
    stDriveMotor := GVL_Motion.AxisDriveMotor,
    stPatchFeedRoll := GVL_Motion.AxisPatchFeedRollMotor,
    stWasteRoll := GVL_Motion.AxisWasteRollMotor
);
GVL_Motion.stPatchFeedStatus := fbPatchFeedManager.stStatus;

// Start-only load policy: two components, or an empty nest when configured.
bOperatorLoadValid :=
    (stInputs.bLoadingStationEaglePresent AND stInputs.bLoadingStationPbupPresent)
    OR (NOT stInputs.bLoadingStationEaglePresent AND NOT stInputs.bLoadingStationPbupPresent
        AND stConfig.bAllowEmptyNestIndex);
fbNestManager.Cyclic(
    bIndexStable := stInputs.bIndexReady AND stInputs.bIndexLocked AND NOT stIndexStatus.bBusy,
    eIndexPosition := stInputs.eIndexPosition,
    eOperatorPosition := stConfig.eOperatorPosition,
    bPartPresent := stInputs.bLoadingStationEaglePresent,
    bPbupPresent := stInputs.bLoadingStationPbupPresent,
    bOperatorReloadPermitted := (eMachineState = E_MachineState.AutoCycle)
        AND ((stOperatorStatus.eState = E_OperatorExchangeState.WaitingForPartLoading)
            OR (stOperatorStatus.eState = E_OperatorExchangeState.ExchangeComplete)),
    aNestEnabled := stConfig.aNestEnabled
);

// =====================================================
// PRODUCTION STATISTICS RESET
// =====================================================
// Reset only the accumulated production counters for
// the selected physical nest.
//
// Test History, current nest data and process results
// are deliberately preserved.

IF (stCommand.uiResetStatisticsNestId >= 1)
    AND (stCommand.uiResetStatisticsNestId <= 4)
THEN

    fbNestManager.ResetNestStatistics(
        uiNestId := stCommand.uiResetStatisticsNestId
    );

END_IF


stOperatorNest := fbNestManager.GetNestAtPosition(stConfig.eOperatorPosition);
stPatchDispenseNest := fbNestManager.GetNestAtPosition(stConfig.ePatchDispensePosition);
stHeatStakeNest := fbNestManager.GetNestAtPosition(stConfig.eHeatStakePosition);
stVisionNest := fbNestManager.GetNestAtPosition(stConfig.eVisionPosition);

// Publish the actual nest currently occupying each process station.
//
// The station nest structures above are already resolved by the
// FB_NestTableManager and are confirmed online to contain the correct nId.
// Use those resolved values directly instead of performing a second
// GetNestIdAtPosition() lookup.
stStatus.uiPatchDispenseNestId := stPatchDispenseNest.nId;
stStatus.uiHeatStakeNestId := stHeatStakeNest.nId;
stStatus.uiVisionNestId := stVisionNest.nId;

aNestSnapshot := fbNestManager.GetAllNests();

bDisabledNestPartPresent := FALSE;
uiDisabledNestPartNestId := 0;

FOR iNestCheck := 1 TO 4 DO
    IF (NOT stConfig.aNestEnabled[iNestCheck])
        AND (aNestSnapshot[iNestCheck].bPartPresent OR aNestSnapshot[iNestCheck].bPbupPresent)
    THEN
        bDisabledNestPartPresent := TRUE;

        IF uiDisabledNestPartNestId = 0 THEN
            uiDisabledNestPartNestId := INT_TO_UINT(iNestCheck);
        END_IF
    END_IF
END_FOR

// A process is required only when:
// - the physical nest contains a part;
// - this stage is still Waiting;
// - every upstream process required for product validity has passed.
//
// This gives deterministic recovery after faults and prevents a failed product
// from being processed by downstream stations.
bPatchDispenseRequired :=
    stPatchDispenseNest.bPartPresent
    AND stPatchDispenseNest.bLoadSetComplete
    AND (stPatchDispenseNest.ePatchDispenseStage = E_NestStageStatus.Waiting);

bHeatStakeRequired :=
    stHeatStakeNest.bPartPresent
    AND stHeatStakeNest.bLoadSetComplete
    AND (stHeatStakeNest.eDisposition <> E_PartDisposition.Reprocess)
    AND (stHeatStakeNest.ePatchDispenseStage = E_NestStageStatus.Complete)
    AND (stHeatStakeNest.eHeatStakeStage = E_NestStageStatus.Waiting);

bVisionRequired :=
    stVisionNest.bPartPresent
    AND stVisionNest.bLoadSetComplete
    AND (stVisionNest.eDisposition <> E_PartDisposition.Reprocess)
    AND (stVisionNest.ePatchDispenseStage = E_NestStageStatus.Complete)
    AND (stVisionNest.eHeatStakeStage = E_NestStageStatus.Complete)
    AND (stVisionNest.eVisionStage = E_NestStageStatus.Waiting);

// Capture active-process state BEFORE station Update(). On Safety loss the
// station FB deliberately goes Disabled in the same scan, so querying IsBusy()
// after Update() would lose the information needed to reject the affected part.
bVisionProcessingBeforeUpdate :=
    (fbVision.IsBusy() OR (bProcessStartStations AND bVisionRequired))
    AND NOT fbVisionManualImages.bActive AND NOT bVisionImageOwnedBeforeUpdate;

fbOperatorStation.Cyclic(bAutomaticActive := (eMachineState = E_MachineState.AutoCycle), bIndexStable := stInputs.bIndexReady AND stInputs.bIndexLocked AND NOT stIndexStatus.bBusy, stOperatorNest := stOperatorNest, bPartPresent := stInputs.bLoadingStationEaglePresent,
    bPbupPresent := stInputs.bLoadingStationPbupPresent, bTwoHandsSafe := stInputs.bTwoHandsSafe,
    bResetRequest := stCommand.bReset, bRejectChutePartPresent := stInputs.bRejectChutePartPresent, bRequireRejectConfirm := TRUE, bAllowEmptyNestIndex := stConfig.bAllowEmptyNestIndex);
stOperatorStatus := fbOperatorStation.GetStatus();

// Acknowledge only this physical nest's warning on the operator's accepted reject edge.
// Reset, stop, fault, sensor recovery and mere part removal do not clear it.
IF stOperatorStatus.bRejectEdgeAccepted
    AND stInputs.bIndexReady AND stInputs.bIndexLocked AND NOT stIndexStatus.bBusy
    AND (stInputs.eIndexPosition <> E_TablePosition.Unknown)
    AND (stOperatorNest.nId >= 1) AND (stOperatorNest.nId <= 4)
    AND stOperatorNest.stHeatStakeResult.bValid
    AND (stOperatorNest.stHeatStakeResult.udiAlertCode = GVL_MASTER.udiHeatStakePatchMissingAlertCode)
THEN
    stHeatStakePresenceResult := stOperatorNest.stHeatStakeResult;
    stHeatStakePresenceResult.udiAlertCode := 0;
    fbNestManager.StoreHeatStakeResultAtPosition(
        ePosition := stConfig.eOperatorPosition,
        stResult := stHeatStakePresenceResult);
END_IF

bPatchStartAllowed := stInputs.bIndexReady AND stInputs.bIndexLocked
    AND NOT stIndexStatus.bBusy AND NOT stCommand.bStop AND NOT stCommand.bReset
    AND NOT stCommand.bManualIndexForward AND NOT stInputs.bEventFault
    AND NOT stInputs.bEventCycleStopRequest AND NOT bRejectChuteStopRequestLatched
    AND NOT bAutoCycleStopRequestLatched AND NOT bProcessRequestIndex
    AND NOT bPatchManualVerticalDownHeld
// TEMP_NO_PATCH_NEST_SUPPORT: original code retained for restoration.
//     AND NOT stCommand.bPatchVerticalUpRequest AND NOT stCommand.bPatchVerticalDownRequest
//     AND NOT stCommand.bPatchSupportExtendRequest AND NOT stCommand.bPatchSupportRetractRequest;
    AND NOT stCommand.bPatchVerticalUpRequest AND NOT stCommand.bPatchVerticalDownRequest;

// Apply the ProcessCycle commands generated on the previous scan.
IF stCommand.bReset OR bProcessCycleCompletePulse THEN
    fbPatchDispense.RequestReset();
    fbHeatStake.RequestReset();
    fbVision.RequestReset();
END_IF

IF (bProcessStopStations OR (eMachineState = E_MachineState.Stopping)
        OR ((eMachineState = E_MachineState.Manual)
            AND (stCommand.bStop OR NOT stCommand.bPatchManualEnable OR bRejectChuteStopRequestLatched)))
    AND fbPatchDispense.IsBusy() THEN
    fbPatchDispense.RequestStop();
END_IF

IF bProcessStopStations THEN
    fbHeatStake.RequestStop();
    fbVision.RequestStop();
END_IF

// Do not apply a previous-scan automatic start after camera RUN is lost.
IF NOT GVL_EtherCAT.stVSKeyenceCamera.bRunStatus THEN
    bProcessStartStations := FALSE;
END_IF

IF bProcessStartStations THEN
    bCycleResultsStored := FALSE;

    IF bPatchDispenseRequired THEN
        IF bPatchStartAllowed THEN fbPatchDispense.RequestStart(); END_IF
    ELSE
        fbNestManager.MarkPatchDispenseNotTestedAtPosition(stConfig.ePatchDispensePosition);
    END_IF

    IF bHeatStakeRequired THEN
        // Product crosscheck at admission, before any Heat Stake sequence is requested.
        IF NOT stInputs.bHeatStakeEaglePresent THEN
            IF (eMachineState = E_MachineState.AutoCycle)
                AND stInputs.stSafety.bSafetyOk
                AND stInputs.bIndexReady AND stInputs.bIndexLocked AND NOT stIndexStatus.bBusy
                AND (stInputs.eIndexPosition <> E_TablePosition.Unknown)
                AND (stHeatStakeNest.nId >= 1) AND (stHeatStakeNest.nId <= 4)
                AND NOT fbHeatStake.IsBusy()
            THEN
                stHeatStakePresenceResult := stEmptyHeatStakePresenceResult;
                stHeatStakePresenceResult.bValid := TRUE;
                stHeatStakePresenceResult.bPassed := FALSE;
                stHeatStakePresenceResult.eCode := E_ProcessResultCode.Fail;
                stHeatStakePresenceResult.udiAlertCode := GVL_MASTER.udiHeatStakePatchMissingAlertCode;
                stHeatStakePresenceResult.sDetail := 'Patch not detected at Heat Stake - Heat FAIL / Vision NOT TESTED';
                fbNestManager.StoreHeatStakeResultAtPosition(
                    ePosition := stConfig.eHeatStakePosition,
                    stResult := stHeatStakePresenceResult);
                FinaliseAndRecordAtPosition(stConfig.eHeatStakePosition);
                // Reclassify immediately so completion/fault handling cannot overwrite this FAIL.
                stHeatStakeNest := fbNestManager.GetNestAtPosition(stConfig.eHeatStakePosition);
                bHeatStakeRequired := FALSE;
            END_IF
        ELSE
            fbHeatStake.RequestStart();
        END_IF
    ELSE
        fbNestManager.MarkHeatStakeNotTestedAtPosition(stConfig.eHeatStakePosition);
    END_IF

    IF bVisionRequired THEN
        fbVision.RequestStart();
    ELSE
        fbNestManager.MarkVisionNotTestedAtPosition(stConfig.eVisionPosition);
    END_IF
END_IF

bPatchManualAllowed :=
    (eMachineState = E_MachineState.Manual)
    AND stCommand.bPatchManualEnable
    AND stInputs.stSafety.bSafetyOk
    AND GVL_Safety.bAirSupplySafe
    AND NOT bRejectChuteStopRequestLatched
    AND bPatchDispenseCommissioned;

// Station 1 nest support removed; legacy support commands have no execution path.

// Detect machine Initialising entry.
// HOME requests are issued once per Initialising sequence.

rtMachineInitialising(
    CLK := (eMachineState = E_MachineState.Initialising)
);

IF rtMachineInitialising.Q THEN
    fbPatchDispense.Home();

    // FUTURE IMPLEMENTATION:
    // fbHeatStake.Home();
    // fbVision.Home();
END_IF

fbPatchDispense.Update(stProcessSettings := GVL_Persistent.stPatchProcessSettings,
    bRunSequenceRequest := stCommand.bPatchManualRunSequence,
    bFeedOnlyRequest := stCommand.bPatchDispenseRequest,
    bStartPermitted := bPatchStartAllowed,
    bHoldUpRequired := bPatchDispenseCommissioned
        AND ((eMachineState = E_MachineState.AutoCycle)
            OR ((eMachineState = E_MachineState.Manual)
                AND (NOT bPatchManualVerticalDownHeld OR stCommand.bIndexerManualEnable OR stIndexStatus.bBusy))
            OR ((eMachineState = E_MachineState.Stopping) AND stIndexStatus.bBusy)),
    bPatchOpticalLeft := stInputs.bPatchOpticalLeft,
    bPatchOpticalRight := stInputs.bPatchOpticalRight,
    // Dispense requires physical UP/DOWN feedback.
    bUseVerticalFeedback := TRUE,
    tVerticalMoveTime := GVL_Motion.stPatchFeedSettings.tPatchVerticalMoveTime,
    bVerticalUpCommand := bPatchVerticalUpCommandPrevious,
    bVerticalDownCommand := bPatchVerticalDownCommandPrevious,
    bVerticalIndexReady => bPatchVerticalIndexReady,
    bVerticalUp := stInputs.bMembraneTransferRetracted,
    bVerticalDown := stInputs.bMembraneTransferExtended,
    bDriveStandstill := GVL_Motion.AxisDriveMotor.bStandstill,
    bDriveBusy := fbPatchFeedManager.stStatus.bDriveBusy,
    bDriveMoving := GVL_Motion.AxisDriveMotor.bMoving,
    bDriveFault := GVL_Motion.AxisDriveMotor.bError,
    bDriveRunRequest => bPatchDriveRunRequest,
    bAirBlowRequest => bPatchSequenceAirRequest,
    bVerticalDownRequest => bPatchSequenceDownRequest,
    bEnable :=
        (
            (eMachineState = E_MachineState.Initialising)
            AND GVL_Safety.bAirSupplySafe
        )
        OR (eMachineState = E_MachineState.ReadyToStart)
        OR (eMachineState = E_MachineState.AutoCycle)
        OR (
            (eMachineState = E_MachineState.Manual)
            AND stCommand.bPatchManualEnable
            AND stInputs.stSafety.bSafetyOk
            AND GVL_Safety.bAirSupplySafe
            AND NOT bRejectChuteStopRequestLatched
            AND bPatchDispenseCommissioned
        ),

    bManualMode :=
        (eMachineState = E_MachineState.Manual),

    // Removed support: compatibility-only pins are ignored by the station FB.
    bManualSupportExtendDesired := FALSE,

    bCommissioned := bPatchDispenseCommissioned,

    bSafetyOk :=
        stInputs.stSafety.bSafetyOk
        AND GVL_Safety.bAirSupplySafe,

    bHomingAllowed :=
        (eMachineState = E_MachineState.Initialising)
        AND GVL_Safety.bAirSupplySafe
        AND stInputs.stSafety.bSafetyOk,

    bSupervisionEnable :=
        (eMachineState = E_MachineState.ReadyToStart)
        OR (eMachineState = E_MachineState.AutoCycle)
        OR (eMachineState = E_MachineState.Manual),

    bReset := stCommand.bReset,

    bSupportRetracted := FALSE,
    bSupportExtended := FALSE,

    tSupportTimeout := T#5S,

    stStatus => stPatchDispenseStatus,

    bVerticalUpRequest =>
        bPatchHomeVerticalUpRequest
);
GVL_HMI.stCommands.bPatchManualRunSequence := FALSE;
GVL_HMI.stCommands.bPatchDispenseRequest := FALSE;
// =====================================================
// PATCH DISPENSING - MANUAL VERTICAL
// =====================================================
// HMI sends one-scan direction requests; retain the selected valve command.
IF NOT bPatchManualAllowed OR NOT stInputs.bMainDoorClosed
    OR stCommand.bStop OR stCommand.bReset OR stInputs.bEventFault
    OR stInputs.bEventCycleStopRequest OR stPatchDispenseStatus.bFault
    OR fbPatchDispense.IsBusy() OR stIndexStatus.bBusy
    OR stCommand.bIndexerManualEnable OR stCommand.bManualIndexForward
    OR bProcessRequestIndex THEN
    bPatchManualVerticalUpHeld := FALSE;
    bPatchManualVerticalDownHeld := FALSE;
ELSIF stCommand.bPatchVerticalUpRequest AND NOT stCommand.bPatchVerticalDownRequest THEN
    bPatchManualVerticalUpHeld := TRUE;
    bPatchManualVerticalDownHeld := FALSE;
ELSIF stCommand.bPatchVerticalDownRequest AND NOT stCommand.bPatchVerticalUpRequest THEN
    bPatchManualVerticalUpHeld := FALSE;
    bPatchManualVerticalDownHeld := TRUE;
ELSIF bPatchManualAllowed
    AND NOT bPatchManualVerticalUpHeld
    AND NOT bPatchManualVerticalDownHeld THEN
    // Re-enable manual control at the default UP direction.
    bPatchManualVerticalUpHeld := TRUE;
END_IF



fbHeatStake.Update(
    bEnable :=
        (eMachineState = E_MachineState.Initialising 
			AND GVL_Safety.bAirSupplySafe)
        OR (eMachineState = E_MachineState.ReadyToStart)
        OR (eMachineState = E_MachineState.AutoCycle)
        OR (eMachineState = E_MachineState.Manual),
    bCommissioned := bHeatStakeCommissioned,
    bSafetyOk := stInputs.stSafety.bSafetyOk,
    bSupervisionEnable := (eMachineState = E_MachineState.ReadyToStart)
        OR (eMachineState = E_MachineState.AutoCycle)
        OR (eMachineState = E_MachineState.Manual),
    bManualMode := (eMachineState = E_MachineState.Manual),
    bReset := stCommand.bReset,
    bSupportRetracted := stInputs.bStation2SupportRetracted,
    bSupportExtended := stInputs.bStation2SupportExtended,
    bHeadUpSensor := stInputs.bHeatStakeHeadUp,
    bHeadDownSensor := stInputs.bHeatStakeHeadDown,
    tSupportTimeout := stConfig.tStationSupportTimeout,
    tHeadMoveTimeout := stConfig.tHeatStakeHeadMoveTimeout,
    stProcessSettings := stHeatStakeProcessSettings,
    stStatus => stHeatStakeStatus,
    bSupportExtendRequest => bStation2SupportExtendRequest,
    bSupportRetractRequest => bStation2SupportRetractRequest,
    bHeadLockRequest => bHeatStakeHeadLockRequest,
    bHeadUnlockRequest => bHeatStakeHeadUnlockRequest,
    bHeadDownRequest => bHeatStakeHeadDownRequest,
    bHeadUpRequest => bHeatStakeHeadUpRequest,
    rPressureCommandBar => rHeatStakePressureCommandBar,
    bContactDwellActive => bHeatStakeContactDwellActive,
    usiSequenceStep => usiHeatStakeSequenceStep,
    bHeadDownTimeoutFault => bHeatStakeStationHeadDownTimeoutFault,
    bHeadUpTimeoutFault => bHeatStakeStationHeadUpTimeoutFault,
    bHeadSensorConflictFault => bHeatStakeStationHeadSensorConflictFault
);

// -------------------------------------------------------------------------
// Heat Stake Manual Mode
// -------------------------------------------------------------------------
rtHeatStakeManualStakePatch(CLK := stCommand.bHeatStakeManualStakePatch);
rtHeatStakeManualUnlock(CLK := stCommand.bHeatStakeManualUnlock);
rtHeatStakeManualLock(CLK := stCommand.bHeatStakeManualLock);
rtHeatStakeManualHeadDown(CLK := stCommand.bHeatStakeManualHeadDown);
rtHeatStakeManualHeadUp(CLK := stCommand.bHeatStakeManualHeadUp);
rtHeatStakeInitialising(CLK := (eMachineState = E_MachineState.Initialising));

IF stCommand.bReset THEN
    bHeatStakeManualHeadDownTimeoutFault := FALSE;
    bHeatStakeManualHeadUpTimeoutFault := FALSE;
END_IF

// System Initialising establishes the known Heat Stake home condition once:
IF rtHeatStakeInitialising.Q THEN
    usiHeatStakeManualActionStep := 100;
    tonHeatStakeManualAction(IN := FALSE);
END_IF

bHeatStakeManualActionBusy := (usiHeatStakeManualActionStep <> 0);

// Manual tooling HOME is based on real feedback.
bHeatStakeManualHomePosition :=
    stInputs.bStation2SupportRetracted
    AND stInputs.bHeatStakeHeadUp
    AND NOT stInputs.bHeatStakeHeadDown
    AND NOT bHeatStakeManualHeadUnlocked
    AND NOT bHeatStakeManualActionBusy;

bHeatStakeManualOutOfHome :=
    (eMachineState = E_MachineState.Manual)
    AND NOT bHeatStakeManualHomePosition;

bHeatStakeManualEnableAllowed :=
    (eMachineState = E_MachineState.Manual)
    AND NOT bRejectChuteStopRequestLatched
    AND stInputs.stSafety.bSafetyOk
    AND NOT fbHeatStake.IsBusy()
    AND NOT bHeatStakeManualActionBusy;

bHeatStakeManualUnlockAllowed :=
    NOT stIndexStatus.bBusy AND NOT stIndexStatus.bTwoHandRequired
    AND NOT stInputs.bTwoHandsSafe AND NOT bManualCameraRecoveryActive
    AND (
    (eMachineState = E_MachineState.Manual)
    AND stCommand.bHeatStakeManualEnable
    AND NOT bRejectChuteStopRequestLatched
    AND stInputs.stSafety.bSafetyOk
    AND NOT fbHeatStake.IsBusy()
    AND NOT bHeatStakeManualActionBusy
    AND NOT bHeatStakeManualHeadUnlocked);

bHeatStakeManualLockAllowed :=
    NOT stIndexStatus.bBusy AND NOT stIndexStatus.bTwoHandRequired
    AND NOT stInputs.bTwoHandsSafe AND NOT bManualCameraRecoveryActive
    AND (
    (eMachineState = E_MachineState.Manual)
    AND stCommand.bHeatStakeManualEnable
    AND NOT bRejectChuteStopRequestLatched
    AND stInputs.stSafety.bSafetyOk
    AND NOT fbHeatStake.IsBusy()
    AND NOT bHeatStakeManualActionBusy
    AND bHeatStakeManualHeadUnlocked);

bHeatStakeManualHeadDownAllowed :=
    NOT stIndexStatus.bBusy AND NOT stIndexStatus.bTwoHandRequired
    AND NOT stInputs.bTwoHandsSafe AND NOT bManualCameraRecoveryActive
    AND (
    (eMachineState = E_MachineState.Manual)
    AND stCommand.bHeatStakeManualEnable
    AND NOT bRejectChuteStopRequestLatched
    AND stInputs.stSafety.bSafetyOk
    AND NOT fbHeatStake.IsBusy()
    AND NOT bHeatStakeManualActionBusy
    AND bHeatStakeManualHeadUnlocked
    AND stInputs.bHeatStakeHeadUp
    AND NOT stInputs.bHeatStakeHeadDown
    // Product protection also applies to a manual DOWN request with a loaded nest.
    AND (NOT stHeatStakeNest.bPartPresent OR stInputs.bHeatStakeEaglePresent)
    AND NOT (stHeatStakeNest.stHeatStakeResult.bValid
        AND (stHeatStakeNest.stHeatStakeResult.udiAlertCode = GVL_MASTER.udiHeatStakePatchMissingAlertCode)));

bHeatStakeManualHeadUpAllowed :=
    NOT stIndexStatus.bBusy AND NOT stIndexStatus.bTwoHandRequired
    AND NOT stInputs.bTwoHandsSafe AND NOT bManualCameraRecoveryActive
    AND (
    (eMachineState = E_MachineState.Manual)
    AND stCommand.bHeatStakeManualEnable
    AND NOT bRejectChuteStopRequestLatched
    AND stInputs.stSafety.bSafetyOk
    AND NOT fbHeatStake.IsBusy()
    AND NOT bHeatStakeManualActionBusy
    AND bHeatStakeManualHeadUnlocked
    AND NOT stInputs.bHeatStakeHeadUp);

bHeatStakeManualSupportAllowed :=
    NOT stIndexStatus.bBusy AND NOT stIndexStatus.bTwoHandRequired
    AND NOT stInputs.bTwoHandsSafe AND NOT bManualCameraRecoveryActive
    AND (
    (eMachineState = E_MachineState.Manual)
    AND stCommand.bHeatStakeManualEnable
    AND stInputs.stSafety.bSafetyOk
    AND NOT fbHeatStake.IsBusy()
    AND NOT bHeatStakeManualActionBusy);
	
	
	
// =====================================================
// PATCH DISPENSING MANUAL MODE - PERMISSIVES
// =====================================================

// General Patch manual enable.
bPatchManualEnableAllowed :=
    (eMachineState = E_MachineState.Manual)
    AND stInputs.stSafety.bSafetyOk
    AND GVL_Safety.bAirSupplySafe
    AND NOT bRejectChuteStopRequestLatched
    AND bPatchDispenseCommissioned;

bPatchManualSupportAllowed :=
    bPatchManualEnableAllowed
    AND stCommand.bPatchManualEnable;
	
	
// =====================================================
// PATCH DISPENSING - MANUAL VERTICAL PERMISSIVES
// =====================================================
bPatchVerticalUpAllowed :=
    bPatchManualEnableAllowed
    AND stCommand.bPatchManualEnable
    AND NOT stCommand.bPatchVerticalDownRequest;

bPatchVerticalDownAllowed :=
    bPatchManualEnableAllowed
    AND stCommand.bPatchManualEnable
    AND NOT stCommand.bPatchVerticalUpRequest;
	

tpPatchAirBlow(
    IN := stCommand.bPatchAirBlowRequest
          AND bPatchManualEnableAllowed
          AND stCommand.bPatchManualEnable AND NOT fbPatchDispense.IsBusy(),
    PT := stconfig.tpPatchAirBlowTimer
);

// TODO: Add physical position and mechanical clearance
// interlocks when Patch Vertical sensors are installed.
// =====================================================
// VISION MANUAL MODE - PERMISSIVES
// =====================================================
// The HMI IsEnabled properties are only operator guidance.
// These PLC permissives are the authority for all Vision manual movement.
//
// Vision Manual Enable itself may only be selected in Manual Mode with
// Safety OK and while no reject-chute controlled stop is active.
bVisionManualEnableAllowed :=
    (eMachineState = E_MachineState.Manual)
    AND stInputs.stSafety.bSafetyOk
    AND NOT bRejectChuteStopRequestLatched
    AND (GVL_EtherCAT.stVSKeyenceCamera.bRunStatus OR bVisionCameraStartBlocked
        OR bManualCameraRecoveryActive OR fbVisionManualImages.bPrepared
        OR (fbVisionManualImages.usiStep = 210) OR fbVisionManualImages.bCameraWarning);
// Run Sequence keeps its separate NOT bVisionCameraStartBlocked admission.
// Manual image recovery must remain operable while the camera reports an error.

// Every individual Vision movement requires the general Vision Enable.
bVisionHorizontalBackAllowed :=
    NOT stIndexStatus.bBusy AND NOT stIndexStatus.bTwoHandRequired
    AND NOT stInputs.bTwoHandsSafe AND NOT bManualCameraRecoveryActive
    AND (
    bVisionManualEnableAllowed
    AND stCommand.bVisionManualEnable
    AND stInputs.bVerticalMiniSlideRetracted);

bVisionHorizontalFrontAllowed :=
    NOT stIndexStatus.bBusy AND NOT stIndexStatus.bTwoHandRequired
    AND NOT stInputs.bTwoHandsSafe AND NOT bManualCameraRecoveryActive
    AND (
    bVisionManualEnableAllowed
    AND stCommand.bVisionManualEnable
    AND stInputs.bVerticalMiniSlideRetracted);

// Full UP is always the recovery direction once Vision manual control is enabled.
bVisionVerticalUpAllowed :=
    NOT stIndexStatus.bBusy AND NOT stIndexStatus.bTwoHandRequired
    AND NOT stInputs.bTwoHandsSafe AND NOT bManualCameraRecoveryActive
    AND (
    bVisionManualEnableAllowed
    AND stCommand.bVisionManualEnable);



// Full DOWN is the pick-side movement.
bVisionVerticalFullDownAllowed :=
    NOT stIndexStatus.bBusy AND NOT stIndexStatus.bTwoHandRequired
    AND NOT stInputs.bTwoHandsSafe AND NOT bManualCameraRecoveryActive
    AND (
    bVisionManualEnableAllowed AND stCommand.bVisionManualEnable
    AND ((stInputs.bHorizontalMiniSlideExtended AND NOT stInputs.bHorizontalMiniSlideRetracted)
        OR (stInputs.bHorizontalMiniSlideRetracted AND NOT stInputs.bHorizontalMiniSlideExtended)));

bVisionGripOpenAllowed :=
    NOT stIndexStatus.bBusy AND NOT stIndexStatus.bTwoHandRequired
    AND NOT stInputs.bTwoHandsSafe AND NOT bManualCameraRecoveryActive
    AND (
    bVisionManualEnableAllowed
    AND stCommand.bVisionManualEnable);

bVisionGripCloseAllowed :=
    NOT stIndexStatus.bBusy AND NOT stIndexStatus.bTwoHandRequired
    AND NOT stInputs.bTwoHandsSafe AND NOT bManualCameraRecoveryActive
    AND (
    bVisionManualEnableAllowed
    AND stCommand.bVisionManualEnable);

bVisionRotate0Allowed :=
    NOT stIndexStatus.bBusy AND NOT stIndexStatus.bTwoHandRequired
    AND NOT stInputs.bTwoHandsSafe AND NOT bManualCameraRecoveryActive
    AND (
    bVisionManualEnableAllowed
    AND stCommand.bVisionManualEnable
    AND stInputs.bVerticalMiniSlideRetracted);

bVisionRotate180Allowed :=
    NOT stIndexStatus.bBusy AND NOT stIndexStatus.bTwoHandRequired
    AND NOT stInputs.bTwoHandsSafe AND NOT bManualCameraRecoveryActive
    AND (
    bVisionManualEnableAllowed
    AND stCommand.bVisionManualEnable
    AND stInputs.bVerticalMiniSlideRetracted);

// Do not use fbVision.IsBusy() here: moving away from the automatic home
// position may make the Vision FB report Busy and would prevent recovery.

	
// RUN SEQUENCE:
// Only allowed from the complete Vision HOME position.
bVisionManualRunSequenceAllowed :=
    NOT stIndexStatus.bBusy AND NOT stIndexStatus.bTwoHandRequired
    AND NOT stInputs.bTwoHandsSafe AND NOT bManualCameraRecoveryActive
    AND (
    NOT fbVisionManualImages.bActive AND NOT fbVisionManualImages.bFault
    AND bVisionManualEnableAllowed
    AND NOT bVisionCameraStartBlocked
    AND stCommand.bVisionManualEnable
    AND stInputs.bHorizontalMiniSlideExtended
    AND stInputs.bVerticalMiniSlideRetracted
    AND stInputs.bRotaryGripperOpened
    AND bVisionRotate0Confirmed
    AND NOT (stVisionNest.stHeatStakeResult.bValid
        AND (stVisionNest.stHeatStakeResult.udiAlertCode = GVL_MASTER.udiHeatStakePatchMissingAlertCode)));
	
	
	// =====================================================
	// VISION MANUAL MODE - HOME PERMISSIVE
	// =====================================================
	
	bVisionManualHomeAllowed :=
    NOT stIndexStatus.bBusy AND NOT stIndexStatus.bTwoHandRequired
    AND NOT stInputs.bTwoHandsSafe AND NOT bManualCameraRecoveryActive
    AND (
        NOT fbVisionManualImages.bActive AND NOT fbVisionManualImages.bFault
		AND bVisionManualEnableAllowed
        AND NOT bVisionCameraStartBlocked
		AND stCommand.bVisionManualEnable
		AND NOT bVisionManualSequenceActive
		AND NOT bVisionManualHomeActive);	

	// =====================================================
	// VISION MANUAL MODE - RUN SEQUENCE REQUEST
	// =====================================================
	
	// Capture the one-scan HMI Run Sequence request.
	IF stCommand.bVisionManualRunSequence
		AND bVisionManualRunSequenceAllowed
		AND NOT bVisionManualSequenceActive
	THEN
		bVisionManualSequenceActive := TRUE;
	END_IF;
	
	
	// Cancel sequence ownership if Manual Mode is left
	// or Vision Manual Enable is removed.
	IF (eMachineState <> E_MachineState.Manual)
		OR NOT bVisionManualEnableAllowed
		OR NOT stCommand.bVisionManualEnable
	THEN
		bVisionManualSequenceActive := FALSE;
	END_IF;
	
	// =====================================================
	// VISION MANUAL MODE - HOME REQUEST
	// =====================================================
	
	// Capture the one-scan HMI Home Position request.
	IF stCommand.bVisionManualHomeRequest
		AND bVisionManualHomeAllowed
		AND NOT bVisionManualHomeActive
	THEN
		bVisionManualHomeActive := TRUE;
	END_IF;
	
	// Cancel Home ownership if Manual Mode is left
	// or Vision Manual Enable is removed.
	IF (eMachineState <> E_MachineState.Manual)
		OR NOT bVisionManualEnableAllowed
		OR NOT stCommand.bVisionManualEnable
	THEN
		bVisionManualHomeActive := FALSE;
	END_IF;

// Manual Mode Stake Pacth allowed permissive
bHeatStakeManualStakeAllowed :=
    NOT stIndexStatus.bBusy AND NOT stIndexStatus.bTwoHandRequired
    AND NOT stInputs.bTwoHandsSafe AND NOT bManualCameraRecoveryActive
    AND (
    (eMachineState = E_MachineState.Manual)
    AND NOT bRejectChuteStopRequestLatched
    AND stCommand.bHeatStakeManualEnable
    AND stInputs.stSafety.bSafetyOk
    AND stHeatStakeTemperatureStatus.bIndexTemperatureReady
    AND fbHeatStake.IsReady()
    AND NOT fbHeatStake.IsBusy()
    AND bHeatStakeManualHomePosition
    AND stInputs.bHeatStakeEaglePresent
    AND NOT (stHeatStakeNest.stHeatStakeResult.bValid
    AND (stHeatStakeNest.stHeatStakeResult.udiAlertCode = GVL_MASTER.udiHeatStakePatchMissingAlertCode))
    AND NOT stIndexStatus.bBusy);
	

// Stake Patch reuses the validated automatic station sequence.
IF rtHeatStakeManualStakePatch.Q AND bHeatStakeManualStakeAllowed THEN
    IF fbHeatStake.RequestStart() THEN
        bHeatStakeManualStakeCycleActive := TRUE;
    END_IF
END_IF

// Return Complete -> Ready automatically after a manual validated cycle.
IF (eMachineState = E_MachineState.Manual)
    AND bHeatStakeManualStakeCycleActive
    AND fbHeatStake.IsDone()
THEN
    fbHeatStake.RequestReset();
    bHeatStakeManualStakeCycleActive := FALSE;
END_IF

// Accept full-course manual actions.
IF rtHeatStakeManualUnlock.Q AND bHeatStakeManualUnlockAllowed THEN
    usiHeatStakeManualActionStep := 10;
    tonHeatStakeManualAction(IN := FALSE);

ELSIF rtHeatStakeManualLock.Q AND bHeatStakeManualLockAllowed THEN
    usiHeatStakeManualActionStep := 20;
    tonHeatStakeManualAction(IN := FALSE);

ELSIF rtHeatStakeManualHeadDown.Q AND bHeatStakeManualHeadDownAllowed THEN
    usiHeatStakeManualActionStep := 30;
    tonHeatStakeManualAction(IN := FALSE);

ELSIF rtHeatStakeManualHeadUp.Q AND bHeatStakeManualHeadUpAllowed THEN
    usiHeatStakeManualActionStep := 40;
    tonHeatStakeManualAction(IN := FALSE);
END_IF

CASE usiHeatStakeManualActionStep OF
    10: // Unlock
        bHeatStakeHeadUnlockRequest := TRUE;
        tonHeatStakeManualAction(IN := TRUE, PT := T#1S);
        IF tonHeatStakeManualAction.Q THEN
            tonHeatStakeManualAction(IN := FALSE);
            bHeatStakeManualHeadUnlocked := TRUE;
            usiHeatStakeManualActionStep := 0;
        END_IF

    20: // Lock
        bHeatStakeHeadLockRequest := TRUE;
        tonHeatStakeManualAction(IN := TRUE, PT := T#1S);
        IF tonHeatStakeManualAction.Q THEN
            tonHeatStakeManualAction(IN := FALSE);
            bHeatStakeManualHeadUnlocked := FALSE;
            usiHeatStakeManualActionStep := 0;
        END_IF

    30: // Head DOWN - real sensor feedback
        bHeatStakeHeadDownRequest := NOT stInputs.bHeatStakeHeadDown;
        rHeatStakePressureCommandBar := stHeatStakeProcessSettings.rDownPressureBar;
        tonHeatStakeManualAction(IN := NOT stInputs.bHeatStakeHeadDown, PT := stConfig.tHeatStakeHeadMoveTimeout);
        IF stInputs.bHeatStakeHeadDown THEN
            tonHeatStakeManualAction(IN := FALSE);
            usiHeatStakeManualActionStep := 0;
        ELSIF tonHeatStakeManualAction.Q THEN
            tonHeatStakeManualAction(IN := FALSE);
            bHeatStakeManualHeadDownTimeoutFault := TRUE;
            usiHeatStakeManualActionStep := 0;
        END_IF

    40: // Head UP - real sensor feedback
        bHeatStakeHeadUpRequest := NOT stInputs.bHeatStakeHeadUp;
        tonHeatStakeManualAction(IN := NOT stInputs.bHeatStakeHeadUp, PT := stConfig.tHeatStakeHeadMoveTimeout);
        IF stInputs.bHeatStakeHeadUp THEN
            tonHeatStakeManualAction(IN := FALSE);
            usiHeatStakeManualActionStep := 0;
        ELSIF tonHeatStakeManualAction.Q THEN
            tonHeatStakeManualAction(IN := FALSE);
            bHeatStakeManualHeadUpTimeoutFault := TRUE;
            usiHeatStakeManualActionStep := 0;
        END_IF

   100: // Initialising: wait for pneumatic supply, then Unlock
    // Do not start any Heat Stake recovery timer until TwinSAFE confirms
    // that pneumatic pressure is physically available.
    IF GVL_Safety.bAirSupplySafe THEN

        bHeatStakeHeadUnlockRequest := TRUE;

        tonHeatStakeManualAction(
            IN := TRUE,
            PT := T#1S
        );

        IF tonHeatStakeManualAction.Q THEN
            tonHeatStakeManualAction(IN := FALSE);

            bHeatStakeManualHeadUnlocked := TRUE;
            usiHeatStakeManualActionStep := 110;
        END_IF

    ELSE
        tonHeatStakeManualAction(IN := FALSE);
    END_IF

	
	110: // Initialising: Head UP - physical feedback required
		// Keep the head unlocked for the complete UP movement.
		IF GVL_Safety.bAirSupplySafe THEN
	
			bHeatStakeHeadUnlockRequest := TRUE;
			bHeatStakeHeadUpRequest := NOT stInputs.bHeatStakeHeadUp;
	
			tonHeatStakeManualAction(
				IN := NOT stInputs.bHeatStakeHeadUp,
				PT := stConfig.tHeatStakeHeadMoveTimeout
			);
	
			IF stInputs.bHeatStakeHeadUp THEN
	
				tonHeatStakeManualAction(IN := FALSE);
				bHeatStakeHeadUpRequest := FALSE;
	
				usiHeatStakeManualActionStep := 120;
	
			ELSIF tonHeatStakeManualAction.Q THEN
	
				tonHeatStakeManualAction(IN := FALSE);
				bHeatStakeManualHeadUpTimeoutFault := TRUE;
	
				usiHeatStakeManualActionStep := 0;
	
			END_IF
	
		ELSE
			// Air disappeared during recovery.
			// Freeze the movement timeout instead of generating a false
			// Head UP timeout while pneumatic movement is impossible.
			bHeatStakeHeadUpRequest := FALSE;
			tonHeatStakeManualAction(IN := FALSE);
		END_IF
	
    120: // Initialising: Lock
        bHeatStakeHeadLockRequest := TRUE;
        tonHeatStakeManualAction(IN := TRUE, PT := T#1S);
        IF tonHeatStakeManualAction.Q THEN
            tonHeatStakeManualAction(IN := FALSE);
            bHeatStakeManualHeadUnlocked := FALSE;
            usiHeatStakeManualActionStep := 130;
        END_IF

    130: // Initialising: Support DOWN
        bStation2SupportRetractRequest := NOT stInputs.bStation2SupportRetracted;
        IF stInputs.bStation2SupportRetracted THEN
            usiHeatStakeManualActionStep := 0;
        END_IF
END_CASE

// Manual UNLOCK is a maintained valve command, not only the 1 s action pulse.
// Leave automatic Stake Patch, homing and fault/recovery ownership unchanged.
IF (eMachineState = E_MachineState.Manual)
    AND NOT bHeatStakeManualStakeCycleActive
    AND NOT fbHeatStake.IsBusy() THEN
    bHeatStakeHeadUnlockRequest :=
        (bHeatStakeHeadUnlockRequest OR bHeatStakeManualHeadUnlocked)
        AND NOT bHeatStakeHeadLockRequest;
END_IF

// Support toggle: ON = UP/Extend, OFF = DOWN/Retract.
// Heat Stake Enable is also required for normal manual support control.
//
// Reject-chute controlled stop:
// if the support was already travelling when the stop request arrived,
// complete that captured target stroke. Do not accept a new target.
IF (eMachineState = E_MachineState.Manual)
    AND bRejectChuteStopRequestLatched
THEN
    IF bManualSupportTargetUpAtRejectStop THEN
        bStation2SupportExtendRequest := NOT stInputs.bStation2SupportExtended;
        bStation2SupportRetractRequest := FALSE;
    ELSE
        bStation2SupportRetractRequest := NOT stInputs.bStation2SupportRetracted;
        bStation2SupportExtendRequest := FALSE;
    END_IF

ELSIF bHeatStakeManualSupportAllowed THEN
    IF stCommand.bHeatStakeManualSupportUp THEN
        bStation2SupportExtendRequest := NOT stInputs.bStation2SupportExtended;
        bStation2SupportRetractRequest := FALSE;
    ELSE
        bStation2SupportRetractRequest := NOT stInputs.bStation2SupportRetracted;
        bStation2SupportExtendRequest := FALSE;
    END_IF
END_IF

// Leaving Manual cancels manual action execution.
// Initialising retains only its dedicated home sequence.
IF (eMachineState <> E_MachineState.Manual)
    AND (eMachineState <> E_MachineState.Initialising)
THEN
    IF usiHeatStakeManualActionStep < 100 THEN
        usiHeatStakeManualActionStep := 0;
        tonHeatStakeManualAction(IN := FALSE);
    END_IF
    bHeatStakeManualStakeCycleActive := FALSE;
END_IF

stHeatStakeProcessStatus.tContactTimeSet 		:= stHeatStakeProcessSettings.tContactTime;
stHeatStakeProcessStatus.rContactTimeSetSeconds := TIME_TO_LREAL(stHeatStakeProcessSettings.tContactTime) / 1000.0;
stHeatStakeProcessStatus.rPressureSetpointBar 	:= stHeatStakeProcessSettings.rDownPressureBar;
stHeatStakeProcessStatus.bHeadLockCommand 		:= bHeatStakeHeadLockRequest;
stHeatStakeProcessStatus.bHeadUnlockCommand 	:= bHeatStakeHeadUnlockRequest;
stHeatStakeProcessStatus.bHeadDownCommand 		:= bHeatStakeHeadDownRequest;
stHeatStakeProcessStatus.bHeadUpCommand 		:= bHeatStakeHeadUpRequest;
stHeatStakeProcessStatus.bContactDwellActive 	:= bHeatStakeContactDwellActive;
stHeatStakeProcessStatus.usiSequenceStep 		:= usiHeatStakeSequenceStep;

// =====================================================
// VISION MANUAL MODE - EXECUTE HOME
// =====================================================

// Generate a single pulse when Home ownership becomes active.
rtVisionManualHome(
    CLK := bVisionManualHomeActive
);

// Request the existing FB_VisionStation controlled homing sequence once.
IF (eMachineState = E_MachineState.Manual)
    AND rtVisionManualHome.Q
THEN
    fbVision.RequestStop();
END_IF;
// =====================================================
// VISION MANUAL MODE - EXECUTE RUN SEQUENCE
// =====================================================

// Start the validated FB_VisionStation sequence.
IF (eMachineState = E_MachineState.Manual)
    AND bVisionManualSequenceActive
    AND NOT fbVision.IsBusy()
    AND NOT fbVision.IsDone()
    AND NOT fbVision.IsFaulted()
    AND NOT (stVisionNest.stHeatStakeResult.bValid
        AND (stVisionNest.stHeatStakeResult.udiAlertCode = GVL_MASTER.udiHeatStakePatchMissingAlertCode))
THEN
    fbVision.RequestStart();
END_IF;


fbVision.Update(stProcessSettings := GVL_Persistent.stVisionProcessSettings,
    // During System Initialising, do not start the Vision homing sequence until
    // TwinSAFE confirms that pneumatic pressure is available. This prevents the
    // station's 5 s tooling-movement timer from expiring while the MS6 / air
    // supply is still being established.
	bEnable :=
		((eMachineState = E_MachineState.Initialising) AND GVL_Safety.bAirSupplySafe)
		OR 	(eMachineState = E_MachineState.ReadyToStart)
		OR 	(eMachineState = E_MachineState.AutoCycle)
		OR 	(
			( eMachineState = E_MachineState.Manual)
			AND ( bVisionManualSequenceActive
			OR bVisionManualHomeActive )
			),
		
    bCommissioned 		:= 	bVisionCommissioned,
    bSafetyOk 			:= 	stInputs.stSafety.bSafetyOk,
    bSupervisionEnable 	:= 	(eMachineState = E_MachineState.ReadyToStart) OR
							(eMachineState = E_MachineState.AutoCycle) OR
        					(eMachineState = E_MachineState.Manual),
							
    bReset := stCommand.bReset,

    bSupportRetracted 	:= FALSE, // Removed hardware; ignored by Vision FB.

    bSupportExtended 	:= FALSE, // Removed hardware; ignored by Vision FB.

    // Mechanical orientation is reversed relative to cylinder naming:
    // EXTENDED = slide BACK (home), RETRACTED = slide FRONT.
    bHorizontalBack 		:= stInputs.bHorizontalMiniSlideExtended,
    bHorizontalFront 		:= stInputs.bHorizontalMiniSlideRetracted,
    bVerticalUp 			:= stInputs.bVerticalMiniSlideRetracted,
    bVerticalDown 			:= stInputs.bVerticalMiniSlideExtended,

    bLimitOff 				:= FALSE, // Removed hardware; ignored by Vision FB.

    bLimitOn 				:= FALSE, // Removed hardware; ignored by Vision FB.
    bGripOpened 			:= stInputs.bRotaryGripperOpened,
    bGripClosed 			:= stInputs.bRotaryGripperClosed,
    bRotate0 				:= bVisionRotate0Confirmed,
    bRotate180 				:= bVisionRotate180Confirmed,
    bRotate0Raw 			:= stInputs.bRotaryGripperPick0,
    bRotate180Raw 			:= stInputs.bRotaryGripperPlace180,
    bCameraTriggerAccepted 	:= bVisionTriggerAccepted,
    bUseOptimizedSequenceTiming := (eMachineState = E_MachineState.AutoCycle)
        OR ((eMachineState = E_MachineState.Manual) AND bVisionManualSequenceActive),
    bCameraReadyForFlip := GVL_EtherCAT.stVSKeyenceCamera.bRunStatus
        AND NOT bVisionCameraStartBlocked
        AND GVL_EtherCAT.stVSKeyenceCamera.bTriggerReady
        AND NOT GVL_EtherCAT.stVSKeyenceCamera.bTriggerAcknowledge
        AND NOT GVL_EtherCAT.stVSKeyenceCamera.bResultsReady
        AND NOT GVL_EtherCAT.stVSKeyenceCamera.bResultAck
        AND NOT GVL_EtherCAT.stVSKeyenceCamera.bProgramLoadExecute,
	
    tSupportTimeout 		:= stConfig.tStationSupportTimeout,
	nCurrentProgramNumber	:= bVisionGetCurrentProgram,
	nVisionCameraResults	:= nVisionResults,
	bResultsReady			:= bVisionGetResultsReadyRequest,

    stStatus 				=> stVisionStatus,

    bHorizontalBackRequest 	=> bVisionHorizontalBackRequest,
    bHorizontalFrontRequest => bVisionHorizontalFrontRequest,
    bVerticalUpRequest 		=> bVisionVerticalUpRequest,
    bVerticalDownRequest 	=> bVisionVerticalDownRequest,

    bGripCloseRequest 		=> bVisionGripCloseRequest,
    bGripOpenRequest 		=> bVisionGripOpenRequest,
    bRotate0Request 		=> bVisionRotate0Request,
    bRotate180Request 		=> bVisionRotate180Request,
	//camera
	bTriggerRequest					=>		bVisionTriggerRequest,
	bChangeProgramRequest			=>		bVisionChangeProgramRequest,
	bGetResultsRequest				=>		bVisionGetResultsRequest,
	bRequestResetResults			=>		bVisionResetResultsRequest,
	bAcknowledgeResults				=> 		bVisionAcknowledgeResultsRquest,
	nProgramNumber					=>		nVisionProgramNumber
);

// Manual image position owner. The automatic station keeps its public contract;
// the following mux arbitrates its requests with the separate manual Vision FB.
bVisionImageOwnedBeforeUpdate := fbVisionManualImages.bActive;
bVisionImageJogBusy := stCommand.bVisionHorizontalBackRequest
    OR stCommand.bVisionHorizontalFrontRequest OR stCommand.bVisionVerticalUpRequest
    OR stCommand.bVisionVerticalFullDownRequest OR stCommand.bVisionGripOpenRequest
    OR stCommand.bVisionGripCloseRequest OR stCommand.bVisionRotate0Request
    OR stCommand.bVisionRotate180Request OR tpVisionManualHorizontalBack.Q
    OR tpVisionManualHorizontalFront.Q OR bVisionManualVerticalUpActive
    OR bVisionManualVerticalFullDownActive OR bVisionManualRotate0Active
    OR bVisionManualRotate180Active;
uiVisionPbupNest := 0;
IF (stInputs.eIndexPosition = E_TablePosition.Unknown) AND NOT stIndexStatus.bBusy THEN
    aVisionPbupReferenceKnown[1] := FALSE;
    aVisionProductLocation[1] := 0;
    aVisionPbupSource[1] := 0;
    aVisionLoadEmptySeen[1] := FALSE;
    aVisionLoadCandidate[1] := FALSE;
    aVisionPbupReferenceKnown[2] := FALSE;
    aVisionProductLocation[2] := 0;
    aVisionPbupSource[2] := 0;
    aVisionLoadEmptySeen[2] := FALSE;
    aVisionLoadCandidate[2] := FALSE;
    aVisionPbupReferenceKnown[3] := FALSE;
    aVisionProductLocation[3] := 0;
    aVisionPbupSource[3] := 0;
    aVisionLoadEmptySeen[3] := FALSE;
    aVisionLoadCandidate[3] := FALSE;
    aVisionPbupReferenceKnown[4] := FALSE;
    aVisionProductLocation[4] := 0;
    aVisionPbupSource[4] := 0;
    aVisionLoadEmptySeen[4] := FALSE;
    aVisionLoadCandidate[4] := FALSE;
END_IF
IF stInputs.bIndexReady AND stInputs.bIndexLocked AND NOT stIndexStatus.bBusy
    AND (stInputs.eIndexPosition <> E_TablePosition.Unknown)
    AND (stVisionNest.nId >= 1) AND (stVisionNest.nId <= 4) THEN
    uiVisionPbupNest := stVisionNest.nId;
END_IF

// Assembly confidence and pickup location belong to the physical product.
// 0=unknown, 1=single nest, 2=legacy alias for nest, 3=held by tooling.
IF (stOperatorNest.nId >= 1) AND (stOperatorNest.nId <= 4)
    AND stInputs.bIndexReady AND stInputs.bIndexLocked AND NOT stIndexStatus.bBusy
    AND (stInputs.eIndexPosition <> E_TablePosition.Unknown) THEN
    IF uiVisionLoadObservedNest <> stOperatorNest.nId THEN
        IF (uiVisionLoadObservedNest >= 1) AND (uiVisionLoadObservedNest <= 4) THEN
            aVisionLoadCandidate[uiVisionLoadObservedNest] := FALSE;
            aVisionLoadEmptySeen[uiVisionLoadObservedNest] := FALSE;
        END_IF
        tonVisionLoadEmpty(IN := FALSE);
        tonVisionLoadPair(IN := FALSE);
        uiVisionLoadObservedNest := stOperatorNest.nId;
    END_IF
    tonVisionLoadEmpty(IN := NOT stInputs.bLoadingStationEaglePresent
        AND NOT stInputs.bLoadingStationPbupPresent, PT := T#200MS);
    tonVisionLoadPair(IN := aVisionLoadCandidate[stOperatorNest.nId]
        AND stInputs.bLoadingStationEaglePresent AND stInputs.bLoadingStationPbupPresent,
        PT := T#200MS);
    IF tonVisionLoadEmpty.Q THEN
        aVisionLoadEmptySeen[stOperatorNest.nId] := TRUE;
        aVisionLoadCandidate[stOperatorNest.nId] := FALSE;
        aVisionPbupReferenceKnown[stOperatorNest.nId] := FALSE;
        aVisionProductLocation[stOperatorNest.nId] := 0;
        aVisionPbupSource[stOperatorNest.nId] := 0;
    END_IF
    IF aVisionLoadEmptySeen[stOperatorNest.nId]
        AND (stInputs.bLoadingStationEaglePresent OR stInputs.bLoadingStationPbupPresent) THEN
        aVisionLoadCandidate[stOperatorNest.nId] := TRUE;
        aVisionLoadEmptySeen[stOperatorNest.nId] := FALSE;
    END_IF
    IF stOperatorNest.bPartLoadedPulse OR stOperatorNest.bPartRemovedPulse THEN
        aVisionPbupReferenceKnown[stOperatorNest.nId] := FALSE;
        aVisionProductLocation[stOperatorNest.nId] := 0;
        aVisionPbupSource[stOperatorNest.nId] := 0;
        IF stOperatorNest.bPartRemovedPulse THEN
            aVisionLoadCandidate[stOperatorNest.nId] := FALSE;
        END_IF
        IF GVL_Persistent.aVisionPbupFitted[stOperatorNest.nId] THEN
            GVL_Persistent.aVisionPbupFitted[stOperatorNest.nId] := FALSE;
            GVL_HMI.bVisionPbupSaveRequest := TRUE;
        END_IF
    END_IF
    IF tonVisionLoadPair.Q AND aVisionLoadCandidate[stOperatorNest.nId] THEN
        aVisionPbupReferenceKnown[stOperatorNest.nId] := TRUE;
        aVisionProductLocation[stOperatorNest.nId] := 1;
        aVisionPbupSource[stOperatorNest.nId] := 1; // Qualified new paired load.
        aVisionLoadCandidate[stOperatorNest.nId] := FALSE;
        GVL_Persistent.aVisionPbupFitted[stOperatorNest.nId] := FALSE;
        GVL_HMI.bVisionPbupSaveRequest := TRUE;
    END_IF
ELSE
    IF (uiVisionLoadObservedNest >= 1) AND (uiVisionLoadObservedNest <= 4) THEN
        aVisionLoadCandidate[uiVisionLoadObservedNest] := FALSE;
        aVisionLoadEmptySeen[uiVisionLoadObservedNest] := FALSE;
    END_IF
    tonVisionLoadEmpty(IN := FALSE);
    tonVisionLoadPair(IN := FALSE);
    uiVisionLoadObservedNest := 0;
END_IF

// Automatic/full manual cycles invalidate confidence at start and establish fitted
// only after a completed cycle. An aborted assembly remains unknown.
rtVisionPbupAutoBusy(CLK := fbVision.IsBusy() AND NOT bVisionImageOwnedBeforeUpdate);
rtVisionPbupAutoDone(CLK := fbVision.IsDone());
IF (uiVisionPbupNest >= 1) AND (uiVisionPbupNest <= 4) THEN
    IF rtVisionPbupAutoBusy.Q THEN
        aVisionPbupReferenceKnown[uiVisionPbupNest] := FALSE;
        aVisionProductLocation[uiVisionPbupNest] := 0;
        aVisionPbupSource[uiVisionPbupNest] := 0;
    END_IF
    IF rtVisionPbupAutoDone.Q THEN
        GVL_Persistent.aVisionPbupFitted[uiVisionPbupNest] := TRUE;
        aVisionPbupReferenceKnown[uiVisionPbupNest] := TRUE;
        aVisionProductLocation[uiVisionPbupNest] := 1;
        aVisionPbupSource[uiVisionPbupNest] := 3;
        GVL_HMI.bVisionPbupFittedEdit := TRUE;
    END_IF
    bVisionPbupFitted := GVL_Persistent.aVisionPbupFitted[uiVisionPbupNest];
    bVisionPbupKnown := aVisionPbupReferenceKnown[uiVisionPbupNest];
    // An old fitted boolean cannot establish a newly unknown pickup location.
    IF aVisionProductLocation[uiVisionPbupNest] = 0 THEN
        aVisionPbupReferenceKnown[uiVisionPbupNest] := FALSE;
        bVisionPbupKnown := FALSE;
    END_IF
ELSE
    bVisionPbupFitted := FALSE;
    bVisionPbupKnown := FALSE;
END_IF

// Checkbox edit buffer is refreshed on nest change and PLC assembly completion.
// A separate confirmation accepts an unchanged FALSE or TRUE value after restart.
IF uiVisionPbupEditNest <> uiVisionPbupNest THEN
    uiVisionPbupEditNest := uiVisionPbupNest;
    GVL_HMI.bVisionPbupFittedEdit := bVisionPbupFitted;

END_IF
GVL_HMI.bVisionPbupEditAllowed := bManualCameraAllowed
    AND NOT bVisionImageOwnedBeforeUpdate AND NOT fbVisionManualImages.bFault
    AND (usiManualCameraStep = 0) AND NOT bVisionImageJogBusy
    AND NOT stCommand.bManualIndexForward AND NOT stCommand.bStop AND NOT stCommand.bReset
    AND (uiVisionPbupNest >= 1) AND (uiVisionPbupNest <= 4)
    AND stVisionStatus.bHome AND stVisionNest.bPartPresent
    AND NOT bManualCameraRecoveryActive;
IF GVL_HMI.bVisionPbupConfirm THEN
    IF GVL_HMI.bVisionPbupEditAllowed THEN
        GVL_Persistent.aVisionPbupFitted[uiVisionPbupNest] := GVL_HMI.bVisionPbupFittedEdit;
        aVisionPbupReferenceKnown[uiVisionPbupNest] := TRUE;
        bVisionPbupFitted := GVL_HMI.bVisionPbupFittedEdit;
        bVisionPbupKnown := TRUE;
        aVisionPbupSource[uiVisionPbupNest] := 2; // Explicit operator confirmation.
        aVisionProductLocation[uiVisionPbupNest] := 1; // The part is in the single nest.
        GVL_HMI.bVisionPbupSaveRequest := TRUE;
    ELSE
        GVL_HMI.bVisionPbupFittedEdit := bVisionPbupFitted;
    END_IF
END_IF
GVL_HMI.bVisionPbupConfirm := FALSE;

bVisionImagePermit := bManualCameraAllowed AND bVisionManualEnableAllowed
    AND NOT fbVision.IsFaulted()
    AND (GVL_HMI.bCameraConnected OR (bVisionImageOwnedBeforeUpdate
        AND (fbVisionManualImages.bPrepared OR (fbVisionManualImages.usiStep = 210))))
    AND (bVisionImageOwnedBeforeUpdate OR NOT bVisionImageJogBusy)
    AND ((uiVisionPbupNest >= 1) AND (uiVisionPbupNest <= 4))
    AND stVisionNest.bPartPresent
    AND (bVisionImageOwnedBeforeUpdate
        OR (NOT bManualCameraRecoveryActive AND NOT stCommand.bManualIndexForward AND NOT stInputs.bTwoHandsSafe
            AND NOT stIndexStatus.bTwoHandRequired AND (fbIndex.GetState() = E_IndexState.Idle)));
IF NOT bVisionImageOwnedBeforeUpdate AND (uiVisionPbupNest >= 1) AND (uiVisionPbupNest <= 4) THEN
    bVisionImagePermit := bVisionImagePermit
        AND ((aVisionProductLocation[uiVisionPbupNest] = 1) OR (aVisionProductLocation[uiVisionPbupNest] = 2));
END_IF
IF NOT bVisionPbupFitted AND (GVL_HMI.udiCameraManualImageSelection <> 1) THEN
    bVisionImagePermit := bVisionImagePermit AND stVisionNest.bLoadSetComplete;
END_IF
IF bVisionImageOwnedBeforeUpdate THEN
    bVisionImagePermit := bVisionImagePermit
        AND (uiVisionPbupNest = uiVisionImageOwnedNest)
        AND (stInputs.eIndexPosition = eVisionImageOwnedIndex);
END_IF

// Retired compatibility symbols: no location selection exists on this machine.
GVL_HMI.bVisionPickupFrontEdit := FALSE;
GVL_HMI.bVisionPickupFrontApplied := FALSE;
fbVisionManualImages(
    bPermit := bVisionImagePermit,
    bReset := stCommand.bReset,
    bPrepare := GVL_HMI.bVisionImagePrepare AND GVL_HMI.bCameraConnected
        AND GVL_EtherCAT.stVSKeyenceCamera.bRunStatus,
    bRelease := GVL_HMI.bVisionImageRelease,
    bTrigger := bManualImageTriggerCommand,
    udiSelection := GVL_HMI.udiCameraManualImageSelection,
    bFitted := bVisionPbupFitted,
    bPickAtFront := FALSE, // Retired compatibility input; pickup derives from PBUP fitted state.
    bReferenceKnown := bVisionPbupKnown,
    bHorizontalBack := stInputs.bHorizontalMiniSlideExtended,
    bHorizontalFront := stInputs.bHorizontalMiniSlideRetracted,
    bVerticalUp := stInputs.bVerticalMiniSlideRetracted,
    bVerticalDown := stInputs.bVerticalMiniSlideExtended,
    bGripOpen := stInputs.bRotaryGripperOpened,
    bGripClosed := stInputs.bRotaryGripperClosed,
    bRotate0 := bVisionRotate0Confirmed,
    bRotate180 := bVisionRotate180Confirmed,
    bRotate0Raw := stInputs.bRotaryGripperPick0,
    bRotate180Raw := stInputs.bRotaryGripperPlace180,
    bCameraReady := bManualCameraTransportReady,
    bCameraAccepted := bVisionTriggerAccepted AND (usiManualCameraStep <> 0),
    bCameraComplete := bManualCameraConsume,
    bCameraFailed := bManualImageCameraFailed,
    bCameraReset := bManualCameraRecoveredPulse,
    bCameraBusy := (usiManualCameraStep <> 0),
    tMovingTriggerDelay := UDINT_TO_TIME(GVL_Persistent.stVisionProcessSettings.udiMovingTriggerDelayMs)
);
GVL_HMI.bVisionImagePrepare := FALSE;
GVL_HMI.bVisionImageRelease := FALSE;
IF fbVisionManualImages.bActive AND NOT bVisionImageOwnedBeforeUpdate THEN
    uiVisionImageOwnedNest := uiVisionPbupNest;
    eVisionImageOwnedIndex := stInputs.eIndexPosition;
END_IF
IF fbVisionManualImages.bReferenceLostPulse THEN
    IF NOT stVisionStatus.bHome THEN bVisionImageRecoveryRequired := TRUE; END_IF
    IF (uiVisionImageOwnedNest >= 1) AND (uiVisionImageOwnedNest <= 4) THEN
        aVisionPbupReferenceKnown[uiVisionImageOwnedNest] := FALSE;
        aVisionProductLocation[uiVisionImageOwnedNest] := 0;
        aVisionPbupSource[uiVisionImageOwnedNest] := 0;
    END_IF
    bVisionPbupKnown := FALSE;
END_IF
IF stVisionStatus.bHome AND NOT fbVisionManualImages.bActive AND NOT fbVisionManualImages.bFault THEN
    bVisionImageRecoveryRequired := FALSE;
END_IF
IF fbVisionManualImages.bFittedPulse AND (uiVisionImageOwnedNest >= 1) AND (uiVisionImageOwnedNest <= 4) THEN
    GVL_Persistent.aVisionPbupFitted[uiVisionImageOwnedNest] := TRUE;
    aVisionPbupReferenceKnown[uiVisionImageOwnedNest] := TRUE;
    aVisionPbupSource[uiVisionImageOwnedNest] := 3;
    bVisionPbupFitted := TRUE;
    bVisionPbupKnown := TRUE;
    GVL_HMI.bVisionPbupFittedEdit := TRUE;
    GVL_HMI.bVisionPbupSaveRequest := TRUE;
END_IF

IF (uiVisionImageOwnedNest >= 1) AND (uiVisionImageOwnedNest <= 4) AND fbVisionManualImages.bActive THEN
    IF fbVisionManualImages.bPartHeld THEN
        aVisionProductLocation[uiVisionImageOwnedNest] := 3;
    ELSIF fbVisionManualImages.bPrepared THEN
        aVisionProductLocation[uiVisionImageOwnedNest] := 1; // Images 1/4 both leave the part in its nest.
    END_IF
END_IF

IF fbVisionManualImages.bActive OR bVisionImageOwnedBeforeUpdate OR fbVisionManualImages.bFault THEN
    bVisionHorizontalBackRequest := fbVisionManualImages.bHorizontalBackRequest;
    bVisionHorizontalFrontRequest := fbVisionManualImages.bHorizontalFrontRequest;
    bVisionVerticalUpRequest := fbVisionManualImages.bVerticalUpRequest;
    bVisionVerticalDownRequest := fbVisionManualImages.bVerticalDownRequest;
    bVisionGripOpenRequest := fbVisionManualImages.bGripOpenRequest;
    bVisionGripCloseRequest := fbVisionManualImages.bGripCloseRequest;
    bVisionRotate0Request := fbVisionManualImages.bRotate0Request;
    bVisionRotate180Request := fbVisionManualImages.bRotate180Request;
END_IF

